C09127=1225.144,417.092,-82.048,-175.674,8.013,148.303
C09128=1225.147,416.687,-81.991,-175.674,8.010,148.302
C09129=1225.154,416.282,-81.934,-175.675,8.006,148.301
C09130=1225.160,415.877,-81.878,-175.676,8.003,148.301
C09131=1225.167,415.473,-81.820,-175.677,7.999,148.300
C09132=1225.171,415.226,-81.786,-175.678,7.997,148.300
C09133=1225.175,414.977,-81.752,-175.678,7.995,148.299
C09134=1225.180,414.730,-81.717,-175.679,7.993,148.299
C09135=1225.184,414.482,-81.682,-175.679,7.991,148.298
C09136=1225.188,414.235,-81.647,-175.679,7.988,148.298
C09137=1225.191,413.987,-81.613,-175.680,7.986,148.298
C09138=1225.196,413.740,-81.578,-175.681,7.985,148.297
C09139=1225.200,413.492,-81.544,-175.681,7.982,148.297
C09140=1225.204,413.244,-81.509,-175.682,7.979,148.296
C09141=1225.207,412.997,-81.474,-175.683,7.977,148.296
C09142=1225.212,412.750,-81.440,-175.683,7.975,148.295
C09143=1225.216,412.502,-81.405,-175.684,7.973,148.295
C09144=1225.220,412.254,-81.370,-175.684,7.971,148.295
C09145=1225.223,412.006,-81.336,-175.684,7.969,148.294
C09146=1225.228,411.759,-81.302,-175.685,7.967,148.294
C09147=1225.233,411.511,-81.267,-175.686,7.964,148.293
C09148=1225.236,411.264,-81.232,-175.686,7.962,148.293
C09149=1225.240,411.017,-81.198,-175.687,7.960,148.293
C09150=1225.244,410.769,-81.163,-175.688,7.958,148.292
C09151=1225.249,410.521,-81.129,-175.688,7.956,148.292
C09152=1225.252,410.274,-81.094,-175.688,7.954,148.291
C09153=1225.256,410.026,-81.060,-175.690,7.951,148.291
C09154=1225.260,409.778,-81.025,-175.690,7.949,148.290
C09155=1225.264,409.531,-80.991,-175.690,7.947,148.290
C09156=1225.269,409.283,-80.957,-175.691,7.945,148.290
C09157=1225.272,409.036,-80.921,-175.691,7.942,148.289
C09158=1225.277,408.789,-80.887,-175.692,7.940,148.289
C09159=1225.280,408.541,-80.852,-175.693,7.938,148.288
C09160=1225.285,408.293,-80.818,-175.693,7.935,148.288
C09161=1225.289,408.045,-80.783,-175.694,7.933,148.288
C09162=1225.293,407.798,-80.749,-175.695,7.931,148.287
C09163=1225.297,407.551,-80.715,-175.695,7.928,148.287
C09164=1225.301,407.303,-80.680,-175.696,7.926,148.286
C09165=1225.305,407.055,-80.646,-175.696,7.924,148.286
C09166=1225.309,406.807,-80.611,-175.697,7.922,148.285
C09167=1225.314,406.560,-80.577,-175.698,7.919,148.285
C09168=1225.317,406.313,-80.543,-175.698,7.917,148.284
C09169=1225.321,406.065,-80.508,-175.699,7.915,148.284
C09170=1225.325,405.818,-80.474,-175.699,7.913,148.284
C09171=1225.329,405.569,-80.439,-175.700,7.910,148.283
C09172=1225.334,405.322,-80.405,-175.701,7.908,148.283
C09173=1225.337,405.074,-80.371,-175.701,7.906,148.282
C09174=1225.342,404.827,-80.336,-175.702,7.904,148.282
C09175=1225.346,404.579,-80.302,-175.703,7.901,148.282
C09176=1225.349,404.332,-80.267,-175.703,7.899,148.281
C09177=1225.354,404.084,-80.233,-175.704,7.897,148.281
C09178=1225.358,403.837,-80.199,-175.705,7.894,148.280
C09179=1225.362,403.589,-80.164,-175.705,7.892,148.280
C09180=1225.366,403.341,-80.130,-175.706,7.889,148.279
C09181=1225.369,403.094,-80.096,-175.707,7.887,148.279
C09182=1225.374,402.846,-80.061,-175.707,7.885,148.279
C09183=1225.378,402.599,-80.027,-175.708,7.882,148.278
C09184=1225.382,402.350,-79.993,-175.709,7.880,148.278
C09185=1225.387,402.103,-79.959,-175.709,7.878,148.277
C09186=1225.391,401.856,-79.925,-175.710,7.875,148.277
C09187=1225.395,401.608,-79.890,-175.711,7.873,148.276
C09188=1225.398,401.361,-79.856,-175.711,7.871,148.276
C09189=1225.402,401.113,-79.821,-175.712,7.868,148.276
C09190=1225.406,400.865,-79.787,-175.713,7.865,148.275
C09191=1225.411,400.618,-79.753,-175.713,7.863,148.275
C09192=1225.415,400.370,-79.718,-175.714,7.861,148.274
C09193=1225.419,400.122,-79.685,-175.715,7.858,148.274
C09194=1225.423,399.875,-79.650,-175.715,7.856,148.273
C09195=1225.427,399.627,-79.616,-175.716,7.854,148.273
C09196=1225.431,399.379,-79.582,-175.717,7.851,148.273
C09197=1225.435,399.132,-79.548,-175.717,7.849,148.272
C09198=1225.439,398.884,-79.513,-175.719,7.846,148.272
C09199=1225.443,398.637,-79.480,-175.719,7.844,148.271
C09200=1225.448,398.389,-79.445,-175.719,7.842,148.271
C09201=1225.451,398.141,-79.411,-175.721,7.839,148.271
C09202=1225.456,397.894,-79.377,-175.721,7.837,148.270
C09203=1225.459,397.647,-79.343,-175.722,7.834,148.270
C09204=1225.464,397.398,-79.309,-175.723,7.832,148.269
C09205=1225.467,397.151,-79.275,-175.724,7.830,148.269
C09206=1225.472,396.904,-79.240,-175.724,7.827,148.268
C09207=1225.475,396.656,-79.206,-175.724,7.825,148.268
C09208=1225.480,396.408,-79.172,-175.726,7.822,148.268
C09209=1225.484,396.161,-79.139,-175.726,7.820,148.267
C09210=1225.489,395.913,-79.104,-175.727,7.817,148.267
C09211=1225.492,395.665,-79.070,-175.728,7.815,148.266
C09212=1225.497,395.417,-79.036,-175.729,7.813,148.266
C09213=1225.500,395.170,-79.002,-175.729,7.810,148.265
C09214=1225.504,394.922,-78.967,-175.730,7.807,148.265
C09215=1225.508,394.675,-78.934,-175.731,7.805,148.265
C09216=1225.513,394.427,-78.900,-175.732,7.803,148.264
C09217=1225.516,394.179,-78.866,-175.732,7.800,148.264
C09218=1225.521,393.932,-78.831,-175.733,7.798,148.263
C09219=1225.525,393.684,-78.798,-175.734,7.796,148.263
C09220=1225.529,393.403,-78.759,-175.735,7.792,148.262
C09221=1225.534,393.120,-78.720,-175.736,7.790,148.262
C09222=1225.539,392.840,-78.682,-175.737,7.787,148.261
C09223=1225.544,392.558,-78.644,-175.738,7.784,148.261
C09224=1225.548,392.310,-78.609,-175.738,7.782,148.261
C09225=1225.551,392.063,-78.575,-175.740,7.779,148.260
C09226=1225.556,391.815,-78.542,-175.740,7.777,148.260
C09227=1225.560,391.567,-78.507,-175.741,7.774,148.259
C09228=1225.563,391.320,-78.473,-175.742,7.772,148.259
C09229=1225.568,391.072,-78.439,-175.743,7.769,148.258
C09230=1225.572,390.824,-78.405,-175.744,7.766,148.258
C09231=1225.576,390.577,-78.372,-175.744,7.764,148.258
C09232=1225.580,390.329,-78.338,-175.745,7.761,148.257
C09233=1225.584,390.081,-78.304,-175.746,7.759,148.257
C09234=1225.589,389.833,-78.270,-175.747,7.756,148.256
C09235=1225.593,389.586,-78.236,-175.748,7.753,148.256
C09236=1225.596,389.338,-78.202,-175.749,7.752,148.256
C09237=1225.601,389.090,-78.168,-175.750,7.748,148.255
C09238=1225.605,388.843,-78.135,-175.750,7.746,148.255
C09239=1225.609,388.596,-78.101,-175.751,7.744,148.254
C09240=1225.613,388.347,-78.067,-175.753,7.741,148.254
C09241=1225.617,388.100,-78.033,-175.753,7.739,148.254
C09242=1225.621,387.852,-78.000,-175.754,7.736,148.253
C09243=1225.626,387.605,-77.965,-175.755,7.733,148.253
C09244=1225.630,387.357,-77.932,-175.756,7.731,148.252
C09245=1225.633,387.109,-77.898,-175.757,7.728,148.252
C09246=1225.638,386.861,-77.864,-175.758,7.725,148.251
C09247=1225.642,386.614,-77.830,-175.759,7.723,148.251
C09248=1225.646,386.366,-77.797,-175.760,7.720,148.251
C09249=1225.650,386.119,-77.763,-175.761,7.718,148.250
C09250=1225.654,385.870,-77.729,-175.762,7.716,148.250
C09251=1225.658,385.623,-77.695,-175.762,7.713,148.249
C09252=1225.662,385.376,-77.662,-175.764,7.710,148.249
C09253=1225.666,385.128,-77.628,-175.764,7.708,148.249
C09254=1225.671,384.880,-77.595,-175.765,7.705,148.248
C09255=1225.674,384.632,-77.561,-175.767,7.702,148.248
C09256=1225.678,384.385,-77.527,-175.767,7.700,148.247
C09257=1225.683,384.137,-77.493,-175.768,7.697,148.247
C09258=1225.687,383.890,-77.460,-175.770,7.694,148.247
C09259=1225.691,383.642,-77.426,-175.771,7.692,148.246
C09260=1225.695,383.394,-77.393,-175.771,7.690,148.246
C09261=1225.699,383.146,-77.358,-175.773,7.687,148.246
C09262=1225.703,382.898,-77.325,-175.774,7.684,148.245
C09263=1225.707,382.651,-77.292,-175.775,7.681,148.245
C09264=1225.711,382.404,-77.258,-175.775,7.679,148.244
C09265=1225.716,382.156,-77.224,-175.777,7.676,148.244
C09266=1225.720,381.908,-77.191,-175.778,7.674,148.244
C09267=1225.723,381.660,-77.157,-175.779,7.671,148.243
C09268=1225.727,381.412,-77.124,-175.780,7.669,148.243
C09269=1225.732,381.165,-77.091,-175.781,7.666,148.242
C09270=1225.736,380.917,-77.056,-175.782,7.663,148.242
C09271=1225.740,380.669,-77.023,-175.783,7.660,148.242
C09272=1225.744,380.422,-76.990,-175.784,7.657,148.241
C09273=1225.749,380.174,-76.957,-175.785,7.655,148.241
C09274=1225.752,379.926,-76.923,-175.786,7.653,148.241
C09275=1225.757,379.678,-76.889,-175.787,7.650,148.240
C09276=1225.761,379.430,-76.856,-175.788,7.647,148.240
C09277=1225.765,379.183,-76.823,-175.790,7.644,148.239
C09278=1225.769,378.936,-76.789,-175.791,7.641,148.239
C09279=1225.773,378.688,-76.756,-175.791,7.639,148.239
C09280=1225.777,378.440,-76.722,-175.793,7.637,148.238
C09281=1225.781,378.192,-76.689,-175.794,7.634,148.238
C09282=1225.786,377.944,-76.655,-175.795,7.631,148.237
C09283=1225.789,377.696,-76.621,-175.796,7.628,148.237
C09284=1225.793,377.449,-76.588,-175.797,7.625,148.237
C09285=1225.798,377.201,-76.555,-175.798,7.622,148.236
C09286=1225.802,376.953,-76.522,-175.800,7.621,148.236
C09287=1225.806,376.706,-76.489,-175.801,7.618,148.236
C09288=1225.810,376.458,-76.455,-175.802,7.615,148.235
C09289=1225.814,376.210,-76.422,-175.803,7.612,148.235
C09290=1225.818,375.963,-76.388,-175.804,7.609,148.234
C09291=1225.823,375.715,-76.355,-175.805,7.607,148.234
C09292=1225.827,375.467,-76.322,-175.807,7.604,148.234
C09293=1225.831,375.219,-76.288,-175.808,7.601,148.233
C09294=1225.835,374.972,-76.255,-175.809,7.598,148.233
C09295=1225.839,374.723,-76.222,-175.811,7.596,148.233
C09296=1225.843,374.476,-76.189,-175.811,7.594,148.232
C09297=1225.847,374.228,-76.155,-175.812,7.591,148.232
C09298=1225.851,373.980,-76.122,-175.814,7.588,148.232
C09299=1225.855,373.732,-76.089,-175.815,7.586,148.231
C09300=1225.859,373.485,-76.056,-175.816,7.583,148.231
C09301=1225.864,373.237,-76.023,-175.818,7.580,148.231
C09302=1225.868,372.989,-75.990,-175.819,7.577,148.230
C09303=1225.872,372.741,-75.956,-175.820,7.575,148.230
C09304=1225.876,372.494,-75.923,-175.821,7.572,148.230
C09305=1225.880,372.246,-75.890,-175.823,7.569,148.229
C09306=1225.884,371.998,-75.857,-175.824,7.566,148.229
C09307=1225.888,371.751,-75.824,-175.825,7.564,148.229
C09308=1225.893,371.503,-75.791,-175.827,7.561,148.228
C09309=1225.897,371.255,-75.757,-175.828,7.558,148.228
C09310=1225.901,371.007,-75.724,-175.829,7.555,148.228
C09311=1225.905,370.760,-75.691,-175.831,7.553,148.227
C09312=1225.909,370.512,-75.658,-175.832,7.550,148.227
C09313=1225.913,370.264,-75.625,-175.833,7.547,148.226
C09314=1225.917,370.016,-75.592,-175.835,7.544,148.226
C09315=1225.922,369.769,-75.559,-175.836,7.542,148.226
C09316=1225.926,369.521,-75.525,-175.837,7.539,148.226
C09317=1225.930,369.273,-75.492,-175.839,7.536,148.225
C09318=1225.934,369.025,-75.460,-175.840,7.533,148.225
C09319=1225.938,368.777,-75.427,-175.841,7.531,148.225
C09320=1225.942,368.530,-75.394,-175.843,7.528,148.224
C09321=1225.946,368.282,-75.361,-175.844,7.525,148.224
C09322=1225.950,368.034,-75.328,-175.845,7.523,148.224
C09323=1225.954,367.787,-75.295,-175.846,7.520,148.223
C09324=1225.959,367.506,-75.258,-175.849,7.516,148.223
C09325=1225.964,367.227,-75.220,-175.850,7.514,148.223
C09326=1225.968,366.947,-75.183,-175.852,7.510,148.222
C09327=1225.973,366.667,-75.146,-175.853,7.507,148.222
C09328=1225.977,366.420,-75.113,-175.854,7.505,148.222
C09329=1225.981,366.173,-75.081,-175.856,7.502,148.221
C09330=1225.985,365.925,-75.047,-175.857,7.499,148.221
C09331=1225.990,365.677,-75.015,-175.859,7.496,148.221
C09332=1225.994,365.429,-74.982,-175.860,7.493,148.220
C09333=1225.998,365.181,-74.949,-175.862,7.490,148.220
C09334=1226.002,364.934,-74.916,-175.863,7.488,148.220
C09335=1226.006,364.685,-74.884,-175.864,7.485,148.219
C09336=1226.010,364.438,-74.851,-175.866,7.482,148.219
C09337=1226.014,364.190,-74.817,-175.868,7.480,148.219
C09338=1226.019,363.941,-74.785,-175.869,7.477,148.219
C09339=1226.023,363.694,-74.752,-175.871,7.475,148.218
C09340=1226.026,363.446,-74.719,-175.872,7.471,148.218
C09341=1226.031,363.198,-74.687,-175.874,7.468,148.218
C09342=1226.035,362.950,-74.654,-175.875,7.465,148.217
C09343=1226.040,362.703,-74.621,-175.877,7.463,148.217
C09344=1226.043,362.455,-74.589,-175.878,7.460,148.217
C09345=1226.047,362.207,-74.556,-175.879,7.458,148.217
C09346=1226.052,361.960,-74.523,-175.881,7.455,148.216
C09347=1226.056,361.711,-74.490,-175.883,7.451,148.216
C09348=1226.059,361.464,-74.458,-175.884,7.449,148.216
C09349=1226.064,361.216,-74.425,-175.886,7.446,148.216
C09350=1226.068,360.968,-74.392,-175.887,7.444,148.215
C09351=1226.072,360.720,-74.360,-175.889,7.441,148.215
C09352=1226.076,360.473,-74.327,-175.890,7.438,148.215
C09353=1226.081,360.225,-74.294,-175.892,7.435,148.214
C09354=1226.085,359.977,-74.262,-175.894,7.432,148.214
C09355=1226.088,359.729,-74.229,-175.895,7.430,148.214
C09356=1226.093,359.481,-74.197,-175.897,7.427,148.214
C09357=1226.097,359.233,-74.164,-175.898,7.424,148.213
C09358=1226.101,358.985,-74.132,-175.900,7.422,148.213
C09359=1226.105,358.738,-74.099,-175.902,7.418,148.213
C09360=1226.110,358.490,-74.067,-175.903,7.416,148.213
C09361=1226.114,358.242,-74.035,-175.905,7.413,148.212
C09362=1226.118,357.994,-74.002,-175.906,7.411,148.212
C09363=1226.122,357.746,-73.969,-175.908,7.408,148.212
C09364=1226.126,357.498,-73.937,-175.910,7.404,148.212
C09365=1226.131,357.251,-73.905,-175.911,7.402,148.211
C09366=1226.135,357.003,-73.871,-175.913,7.399,148.211
C09367=1226.138,356.755,-73.840,-175.914,7.397,148.211
C09368=1226.143,356.506,-73.807,-175.916,7.394,148.211
C09369=1226.147,356.259,-73.774,-175.918,7.391,148.210
C09370=1226.151,356.011,-73.742,-175.920,7.388,148.210
C09371=1226.156,355.763,-73.710,-175.921,7.386,148.210
C09372=1226.159,355.516,-73.677,-175.922,7.383,148.210
C09373=1226.164,355.267,-73.645,-175.924,7.380,148.210
C09374=1226.168,355.020,-73.612,-175.926,7.377,148.209
C09375=1226.172,354.772,-73.580,-175.928,7.374,148.209
C09376=1226.177,354.524,-73.548,-175.930,7.372,148.209
C09377=1226.180,354.276,-73.516,-175.931,7.369,148.209
C09378=1226.184,354.028,-73.483,-175.933,7.366,148.208
C09379=1226.189,353.781,-73.451,-175.935,7.363,148.208
C09380=1226.193,353.532,-73.419,-175.936,7.361,148.208
C09381=1226.197,353.284,-73.387,-175.938,7.358,148.208
C09382=1226.201,353.037,-73.354,-175.939,7.356,148.208
C09383=1226.205,352.789,-73.323,-175.942,7.352,148.207
C09384=1226.210,352.541,-73.290,-175.943,7.350,148.207
C09385=1226.213,352.293,-73.258,-175.945,7.347,148.207
C09386=1226.218,352.045,-73.225,-175.947,7.345,148.207
C09387=1226.222,351.798,-73.194,-175.949,7.341,148.207
C09388=1226.226,351.550,-73.161,-175.950,7.338,148.206
C09389=1226.230,351.301,-73.129,-175.951,7.336,148.206
C09390=1226.234,351.053,-73.097,-175.953,7.333,148.206
C09391=1226.239,350.806,-73.065,-175.955,7.330,148.206
C09392=1226.243,350.558,-73.032,-175.957,7.327,148.205
C09393=1226.247,350.310,-73.000,-175.959,7.325,148.205
C09394=1226.252,350.062,-72.968,-175.960,7.322,148.205
C09395=1226.255,349.814,-72.936,-175.962,7.319,148.205
C09396=1226.260,349.566,-72.904,-175.964,7.317,148.205
C09397=1226.264,349.319,-72.873,-175.966,7.314,148.204
C09398=1226.269,349.070,-72.840,-175.967,7.311,148.204
C09399=1226.272,348.822,-72.808,-175.969,7.308,148.204
C09400=1226.276,348.574,-72.776,-175.971,7.306,148.204
C09401=1226.281,348.327,-72.744,-175.973,7.303,148.204
C09402=1226.285,348.079,-72.713,-175.974,7.301,148.203
C09403=1226.289,347.830,-72.680,-175.976,7.297,148.203
C09404=1226.294,347.583,-72.649,-175.979,7.295,148.203
C09405=1226.297,347.335,-72.617,-175.980,7.292,148.203
C09406=1226.302,347.087,-72.585,-175.982,7.289,148.203
C09407=1226.306,346.839,-72.553,-175.984,7.287,148.203
C09408=1226.310,346.591,-72.521,-175.986,7.284,148.202
C09409=1226.315,346.343,-72.489,-175.987,7.281,148.202
C09410=1226.318,346.095,-72.457,-175.989,7.278,148.202
C09411=1226.322,345.847,-72.425,-175.991,7.276,148.202
C09412=1226.327,345.600,-72.393,-175.993,7.273,148.202
C09413=1226.331,345.352,-72.361,-175.995,7.270,148.201
C09414=1226.335,345.104,-72.329,-175.997,7.267,148.202
C09415=1226.340,344.856,-72.297,-175.999,7.265,148.201
C09416=1226.343,344.608,-72.266,-176.000,7.262,148.201
C09417=1226.348,344.361,-72.234,-176.002,7.259,148.201
C09418=1226.352,344.112,-72.202,-176.004,7.256,148.201
C09419=1226.356,343.864,-72.170,-176.006,7.254,148.201
C09420=1226.360,343.616,-72.139,-176.008,7.251,148.200
C09421=1226.365,343.368,-72.107,-176.010,7.248,148.200
C09422=1226.369,343.121,-72.075,-176.012,7.246,148.200
C09423=1226.373,342.873,-72.043,-176.013,7.243,148.200
C09424=1226.377,342.625,-72.011,-176.015,7.240,148.200
C09425=1226.382,342.376,-71.980,-176.017,7.237,148.200
C09426=1226.386,342.128,-71.948,-176.019,7.235,148.200
C09427=1226.390,341.881,-71.917,-176.021,7.232,148.199
C09428=1226.394,341.603,-71.881,-176.023,7.229,148.199
C09429=1226.400,341.325,-71.846,-176.025,7.226,148.199
C09430=1226.404,341.047,-71.810,-176.028,7.223,148.199
C09431=1226.409,340.770,-71.775,-176.029,7.220,148.199
C09432=1226.413,340.522,-71.744,-176.032,7.217,148.199
C09433=1226.417,340.274,-71.712,-176.033,7.214,148.198
C09434=1226.422,340.026,-71.680,-176.035,7.212,148.198
C09435=1226.426,339.778,-71.649,-176.037,7.209,148.198
C09436=1226.430,339.530,-71.617,-176.039,7.206,148.198
C09437=1226.434,339.282,-71.585,-176.041,7.204,148.198
C09438=1226.438,339.034,-71.555,-176.043,7.201,148.198
C09439=1226.442,338.786,-71.523,-176.045,7.198,148.198
C09440=1226.447,338.538,-71.492,-176.047,7.196,148.197
C09441=1226.451,338.290,-71.459,-176.049,7.193,148.197
C09442=1226.455,338.043,-71.428,-176.051,7.190,148.197
C09443=1226.459,337.794,-71.397,-176.053,7.188,148.197
C09444=1226.464,337.547,-71.365,-176.055,7.185,148.197
C09445=1226.468,337.298,-71.334,-176.057,7.182,148.197
C09446=1226.472,337.051,-71.303,-176.059,7.180,148.197
C09447=1226.476,336.802,-71.271,-176.061,7.177,148.197
C09448=1226.480,336.555,-71.240,-176.063,7.174,148.197
C09449=1226.484,336.306,-71.208,-176.065,7.172,148.197
C09450=1226.489,336.059,-71.178,-176.066,7.169,148.196
C09451=1226.492,335.810,-71.146,-176.069,7.166,148.196
C09452=1226.497,335.563,-71.115,-176.071,7.164,148.196
C09453=1226.501,335.314,-71.083,-176.072,7.161,148.196
C09454=1226.506,335.066,-71.052,-176.075,7.158,148.196
C09455=1226.510,334.818,-71.020,-176.077,7.155,148.196
C09456=1226.514,334.570,-70.989,-176.078,7.153,148.196
C09457=1226.518,334.322,-70.958,-176.081,7.150,148.196
C09458=1226.523,334.074,-70.927,-176.083,7.147,148.195
C09459=1226.527,333.826,-70.896,-176.085,7.145,148.195
C09460=1226.531,333.578,-70.864,-176.087,7.142,148.195
C09461=1226.536,333.330,-70.833,-176.089,7.139,148.195
C09462=1226.540,333.082,-70.802,-176.091,7.137,148.195
C09463=1226.544,332.834,-70.771,-176.093,7.134,148.195
C09464=1226.547,332.586,-70.740,-176.095,7.131,148.195
C09465=1226.551,332.339,-70.709,-176.096,7.129,148.195
C09466=1226.556,332.091,-70.678,-176.099,7.126,148.195
C09467=1226.560,331.842,-70.647,-176.101,7.123,148.195
C09468=1226.564,331.595,-70.615,-176.103,7.121,148.195
C09469=1226.568,331.346,-70.584,-176.105,7.118,148.194
C09470=1226.573,331.098,-70.553,-176.107,7.115,148.194
C09471=1226.578,330.850,-70.522,-176.109,7.113,148.194
C09472=1226.581,330.602,-70.491,-176.111,7.110,148.194
C09473=1226.586,330.354,-70.460,-176.113,7.107,148.194
C09474=1226.590,330.105,-70.429,-176.115,7.105,148.194
C09475=1226.595,329.857,-70.398,-176.117,7.102,148.194
C09476=1226.599,329.610,-70.366,-176.119,7.099,148.194
C09477=1226.602,329.362,-70.336,-176.121,7.097,148.194
C09478=1226.607,329.114,-70.305,-176.124,7.094,148.194
C09479=1226.611,328.866,-70.274,-176.126,7.092,148.194
C09480=1226.615,328.618,-70.243,-176.127,7.089,148.194
C09481=1226.620,328.370,-70.212,-176.130,7.086,148.194
C09482=1226.624,328.122,-70.181,-176.132,7.084,148.193
C09483=1226.628,327.873,-70.150,-176.134,7.081,148.193
C09484=1226.632,327.626,-70.120,-176.136,7.078,148.193
C09485=1226.637,327.378,-70.089,-176.138,7.076,148.193
C09486=1226.641,327.129,-70.058,-176.140,7.074,148.193
C09487=1226.645,326.882,-70.026,-176.142,7.070,148.193
C09488=1226.650,326.634,-69.996,-176.144,7.068,148.193
C09489=1226.653,326.385,-69.965,-176.147,7.066,148.193
C09490=1226.658,326.137,-69.934,-176.149,7.062,148.193
C09491=1226.662,325.889,-69.904,-176.151,7.060,148.193
C09492=1226.666,325.641,-69.872,-176.152,7.058,148.193
C09493=1226.670,325.393,-69.842,-176.155,7.055,148.193
C09494=1226.675,325.145,-69.811,-176.157,7.052,148.193
C09495=1226.679,324.896,-69.780,-176.159,7.050,148.193
C09496=1226.683,324.649,-69.750,-176.161,7.047,148.193
C09497=1226.687,324.401,-69.719,-176.164,7.044,148.193
C09498=1226.692,324.153,-69.689,-176.165,7.042,148.193
C09499=1226.696,323.904,-69.658,-176.168,7.039,148.193
C09500=1226.700,323.657,-69.627,-176.170,7.037,148.193
C09501=1226.704,323.409,-69.597,-176.172,7.034,148.192
C09502=1226.709,323.161,-69.566,-176.174,7.031,148.192
C09503=1226.713,322.912,-69.535,-176.176,7.029,148.192
C09504=1226.717,322.664,-69.505,-176.178,7.027,148.193
C09505=1226.721,322.416,-69.474,-176.181,7.023,148.192
C09506=1226.726,322.168,-69.443,-176.183,7.021,148.192
C09507=1226.730,321.919,-69.413,-176.185,7.019,148.192
C09508=1226.734,321.672,-69.382,-176.187,7.015,148.192
C09509=1226.738,321.424,-69.352,-176.189,7.013,148.192
C09510=1226.743,321.176,-69.322,-176.191,7.011,148.192
C09511=1226.747,320.927,-69.290,-176.194,7.008,148.192
C09512=1226.751,320.680,-69.260,-176.196,7.005,148.192
C09513=1226.756,320.431,-69.230,-176.198,7.003,148.192
C09514=1226.760,320.183,-69.199,-176.200,7.000,148.192
C09515=1226.763,319.935,-69.169,-176.202,6.998,148.192
C09516=1226.768,319.687,-69.138,-176.204,6.995,148.192
C09517=1226.772,319.439,-69.108,-176.207,6.992,148.192
C09518=1226.777,319.191,-69.078,-176.209,6.990,148.192
C09519=1226.781,318.943,-69.048,-176.211,6.988,148.192
C09520=1226.785,318.695,-69.017,-176.214,6.985,148.192
C09521=1226.789,318.446,-68.986,-176.215,6.982,148.192
C09522=1226.794,318.198,-68.956,-176.217,6.980,148.192
C09523=1226.798,317.950,-68.926,-176.220,6.977,148.192
C09524=1226.802,317.702,-68.895,-176.222,6.975,148.192
C09525=1226.807,317.454,-68.865,-176.224,6.973,148.192
C09526=1226.811,317.206,-68.835,-176.226,6.969,148.192
C09527=1226.815,316.958,-68.804,-176.228,6.967,148.192
C09528=1226.819,316.709,-68.775,-176.230,6.965,148.192
C09529=1226.824,316.461,-68.744,-176.233,6.962,148.192
C09530=1226.828,316.214,-68.714,-176.235,6.960,148.192
C09531=1226.832,315.965,-68.684,-176.237,6.957,148.192
C09532=1226.836,315.690,-68.650,-176.240,6.954,148.192
C09533=1226.842,315.413,-68.616,-176.242,6.951,148.192
C09534=1226.846,315.138,-68.583,-176.245,6.948,148.192
C09535=1226.851,314.862,-68.550,-176.247,6.946,148.192
C09536=1226.855,314.614,-68.519,-176.250,6.943,148.192
C09537=1226.860,314.366,-68.489,-176.252,6.940,148.192
C09538=1226.864,314.118,-68.459,-176.254,6.938,148.192
C09539=1226.868,313.869,-68.429,-176.256,6.935,148.192
C09540=1226.872,313.621,-68.399,-176.259,6.933,148.192
C09541=1226.876,313.373,-68.369,-176.261,6.931,148.192
C09542=1226.881,313.125,-68.338,-176.263,6.928,148.192
C09543=1226.885,312.877,-68.309,-176.265,6.925,148.192
C09544=1226.890,312.629,-68.278,-176.267,6.923,148.192
C09545=1226.894,312.381,-68.249,-176.270,6.920,148.192
C09546=1226.898,312.133,-68.218,-176.272,6.917,148.192
C09547=1226.903,311.884,-68.188,-176.274,6.915,148.192
C09548=1226.907,311.637,-68.158,-176.277,6.912,148.192
C09549=1226.911,311.388,-68.129,-176.279,6.910,148.192
C09550=1226.916,311.140,-68.099,-176.281,6.908,148.192
C09551=1226.920,310.892,-68.069,-176.283,6.906,148.192
C09552=1226.924,310.644,-68.039,-176.286,6.902,148.192
C09553=1226.929,310.395,-68.009,-176.288,6.900,148.192
C09554=1226.933,310.148,-67.979,-176.290,6.898,148.192
C09555=1226.936,309.899,-67.949,-176.292,6.895,148.192
C09556=1226.941,309.650,-67.919,-176.295,6.893,148.192
C09557=1226.945,309.402,-67.889,-176.297,6.891,148.192
C09558=1226.949,309.154,-67.859,-176.299,6.887,148.192
C09559=1226.954,308.906,-67.829,-176.301,6.885,148.192
C09560=1226.958,308.658,-67.799,-176.303,6.883,148.192
C09561=1226.962,308.410,-67.770,-176.306,6.880,148.192
C09562=1226.966,308.161,-67.740,-176.308,6.878,148.193
C09563=1226.971,307.913,-67.710,-176.310,6.876,148.193
C09564=1226.975,307.665,-67.680,-176.313,6.873,148.193
C09565=1226.979,307.417,-67.651,-176.315,6.870,148.193
C09566=1226.984,307.169,-67.622,-176.317,6.868,148.193
C09567=1226.989,306.921,-67.592,-176.320,6.865,148.193
C09568=1226.993,306.673,-67.562,-176.322,6.863,148.193
C09569=1226.997,306.425,-67.532,-176.324,6.861,148.193
C09570=1227.001,306.177,-67.502,-176.327,6.858,148.193
C09571=1227.005,305.928,-67.473,-176.329,6.855,148.193
C09572=1227.010,305.680,-67.443,-176.331,6.853,148.193
C09573=1227.014,305.431,-67.413,-176.333,6.851,148.193
C09574=1227.019,305.183,-67.384,-176.336,6.848,148.193
C09575=1227.023,304.935,-67.355,-176.338,6.846,148.193
C09576=1227.027,304.687,-67.324,-176.340,6.843,148.193
C09577=1227.031,304.439,-67.295,-176.343,6.840,148.193
C09578=1227.035,304.191,-67.266,-176.345,6.838,148.193
C09579=1227.040,303.942,-67.235,-176.347,6.836,148.193
C09580=1227.044,303.694,-67.206,-176.350,6.833,148.193
C09581=1227.048,303.446,-67.177,-176.352,6.831,148.193
C09582=1227.053,303.198,-67.147,-176.354,6.829,148.194
C09583=1227.057,302.950,-67.118,-176.356,6.826,148.194
C09584=1227.062,302.702,-67.089,-176.359,6.823,148.194
C09585=1227.066,302.453,-67.059,-176.361,6.821,148.194
C09586=1227.070,302.205,-67.030,-176.363,6.819,148.194
C09587=1227.074,301.957,-67.000,-176.366,6.816,148.194
C09588=1227.078,301.708,-66.971,-176.368,6.814,148.194
C09589=1227.082,301.460,-66.941,-176.370,6.812,148.194
C09590=1227.087,301.212,-66.911,-176.373,6.809,148.194
C09591=1227.092,300.964,-66.882,-176.375,6.807,148.194
C09592=1227.096,300.716,-66.853,-176.377,6.804,148.194
C09593=1227.101,300.467,-66.824,-176.379,6.802,148.194
C09594=1227.105,300.219,-66.795,-176.382,6.799,148.194
C09595=1227.109,299.970,-66.765,-176.384,6.797,148.194
C09596=1227.113,299.722,-66.736,-176.386,6.795,148.194
C09597=1227.118,299.474,-66.706,-176.389,6.792,148.195
C09598=1227.122,299.226,-66.677,-176.392,6.790,148.195
C09599=1227.126,298.978,-66.648,-176.394,6.787,148.195
C09600=1227.131,298.729,-66.619,-176.396,6.785,148.195
C09601=1227.135,298.481,-66.589,-176.398,6.782,148.195
C09602=1227.139,298.233,-66.560,-176.401,6.780,148.195
C09603=1227.143,297.985,-66.531,-176.403,6.778,148.195
C09604=1227.148,297.737,-66.502,-176.406,6.775,148.195
C09605=1227.152,297.488,-66.473,-176.408,6.773,148.195
C09606=1227.156,297.240,-66.444,-176.410,6.771,148.195
C09607=1227.160,296.992,-66.414,-176.412,6.768,148.195
C09608=1227.165,296.743,-66.385,-176.415,6.766,148.196
C09609=1227.170,296.495,-66.357,-176.417,6.763,148.196
C09610=1227.174,296.247,-66.327,-176.419,6.761,148.196
C09611=1227.178,295.999,-66.298,-176.422,6.758,148.196
C09612=1227.183,295.750,-66.269,-176.424,6.756,148.196
C09613=1227.187,295.503,-66.240,-176.427,6.754,148.196
C09614=1227.191,295.254,-66.211,-176.429,6.752,148.196
C09615=1227.195,295.005,-66.182,-176.432,6.749,148.196
C09616=1227.199,294.757,-66.153,-176.434,6.746,148.196
C09617=1227.204,294.510,-66.124,-176.436,6.745,148.196
C09618=1227.209,294.261,-66.095,-176.438,6.742,148.196
C09619=1227.213,294.012,-66.065,-176.441,6.739,148.196
C09620=1227.216,293.764,-66.037,-176.443,6.737,148.197
C09621=1227.221,293.516,-66.008,-176.446,6.735,148.197
C09622=1227.226,293.268,-65.979,-176.448,6.733,148.197
C09623=1227.230,293.019,-65.950,-176.451,6.730,148.197
C09624=1227.234,292.771,-65.921,-176.453,6.728,148.197
C09625=1227.239,292.523,-65.893,-176.455,6.726,148.197
C09626=1227.243,292.275,-65.863,-176.458,6.723,148.197
C09627=1227.247,292.026,-65.835,-176.460,6.721,148.197
C09628=1227.252,291.778,-65.806,-176.462,6.718,148.197
C09629=1227.256,291.530,-65.777,-176.465,6.716,148.198
C09630=1227.260,291.281,-65.748,-176.467,6.713,148.198
C09631=1227.264,291.032,-65.719,-176.470,6.711,148.198
C09632=1227.269,290.785,-65.690,-176.472,6.709,148.198
C09633=1227.273,290.536,-65.662,-176.474,6.707,148.198
C09634=1227.277,290.288,-65.633,-176.477,6.704,148.198
C09635=1227.282,290.040,-65.604,-176.479,6.702,148.198
C09636=1227.287,289.766,-65.573,-176.482,6.700,148.198
C09637=1227.292,289.492,-65.540,-176.484,6.697,148.198
C09638=1227.296,289.217,-65.509,-176.487,6.694,148.199
C09639=1227.301,288.943,-65.477,-176.489,6.692,148.199
C09640=1227.306,288.695,-65.449,-176.492,6.690,148.199
C09641=1227.310,288.447,-65.420,-176.495,6.687,148.199
C09642=1227.315,288.199,-65.391,-176.497,6.685,148.199
C09643=1227.319,287.950,-65.363,-176.499,6.683,148.199
C09644=1227.323,287.702,-65.334,-176.502,6.681,148.199
C09645=1227.327,287.454,-65.306,-176.504,6.678,148.199
C09646=1227.332,287.205,-65.277,-176.507,6.676,148.200
C09647=1227.336,286.957,-65.248,-176.509,6.673,148.200
C09648=1227.340,286.709,-65.220,-176.511,6.671,148.200
C09649=1227.345,286.460,-65.191,-176.514,6.669,148.200
C09650=1227.350,286.212,-65.163,-176.516,6.666,148.200
C09651=1227.353,285.964,-65.134,-176.518,6.664,148.200
C09652=1227.358,285.715,-65.105,-176.521,6.662,148.201
C09653=1227.362,285.467,-65.077,-176.523,6.660,148.201
C09654=1227.366,285.218,-65.049,-176.526,6.657,148.201
C09655=1227.371,284.970,-65.021,-176.528,6.655,148.201
C09656=1227.375,284.722,-64.991,-176.530,6.653,148.201
C09657=1227.379,284.473,-64.963,-176.533,6.651,148.201
C09658=1227.384,284.225,-64.935,-176.535,6.649,148.201
C09659=1227.388,283.977,-64.906,-176.538,6.646,148.201
C09660=1227.393,283.729,-64.878,-176.540,6.644,148.202
C09661=1227.397,283.480,-64.850,-176.543,6.641,148.202
C09662=1227.401,283.232,-64.822,-176.545,6.640,148.202
C09663=1227.406,282.983,-64.793,-176.548,6.637,148.202
C09664=1227.410,282.736,-64.765,-176.550,6.634,148.202
C09665=1227.415,282.487,-64.736,-176.553,6.632,148.202
C09666=1227.419,282.239,-64.708,-176.555,6.630,148.202
C09667=1227.423,281.990,-64.679,-176.557,6.628,148.203
C09668=1227.428,281.742,-64.652,-176.560,6.625,148.203
C09669=1227.432,281.493,-64.623,-176.562,6.623,148.203
C09670=1227.436,281.245,-64.595,-176.565,6.621,148.203
C09671=1227.440,280.997,-64.567,-176.567,6.619,148.203
C09672=1227.445,280.748,-64.538,-176.569,6.617,148.203
C09673=1227.449,280.500,-64.511,-176.572,6.614,148.203
C09674=1227.454,280.251,-64.482,-176.575,6.612,148.204
C09675=1227.458,280.003,-64.454,-176.577,6.610,148.204
C09676=1227.462,279.755,-64.426,-176.579,6.608,148.204
C09677=1227.467,279.507,-64.397,-176.581,6.606,148.204
C09678=1227.471,279.259,-64.370,-176.584,6.603,148.204
C09679=1227.476,279.010,-64.341,-176.587,6.601,148.204
C09680=1227.480,278.761,-64.314,-176.589,6.599,148.205
C09681=1227.484,278.513,-64.286,-176.591,6.597,148.205
C09682=1227.489,278.265,-64.257,-176.593,6.594,148.205
C09683=1227.493,278.016,-64.229,-176.596,6.593,148.205
C09684=1227.497,277.768,-64.201,-176.599,6.590,148.205
C09685=1227.502,277.519,-64.173,-176.601,6.588,148.206
C09686=1227.506,277.271,-64.145,-176.603,6.585,148.206
C09687=1227.510,277.022,-64.118,-176.606,6.584,148.206
C09688=1227.515,276.774,-64.089,-176.608,6.581,148.206
C09689=1227.520,276.526,-64.061,-176.611,6.579,148.206
C09690=1227.523,276.278,-64.033,-176.613,6.576,148.206
C09691=1227.528,276.029,-64.005,-176.616,6.574,148.207
C09692=1227.532,275.780,-63.977,-176.618,6.572,148.207
C09693=1227.537,275.532,-63.950,-176.621,6.570,148.207
C09694=1227.541,275.284,-63.922,-176.623,6.568,148.207
C09695=1227.546,275.036,-63.893,-176.626,6.565,148.207
C09696=1227.550,274.787,-63.866,-176.628,6.563,148.207
C09697=1227.554,274.538,-63.838,-176.631,6.561,148.208
C09698=1227.558,274.291,-63.810,-176.633,6.559,148.208
C09699=1227.563,274.042,-63.781,-176.635,6.557,148.208
C09700=1227.568,273.793,-63.754,-176.638,6.555,148.208
C09701=1227.572,273.545,-63.727,-176.641,6.552,148.208
C09702=1227.576,273.297,-63.698,-176.643,6.550,148.208
C09703=1227.581,273.048,-63.671,-176.645,6.548,148.209
C09704=1227.585,272.800,-63.643,-176.648,6.546,148.209
C09705=1227.589,272.551,-63.616,-176.650,6.544,148.209
C09706=1227.594,272.303,-63.588,-176.652,6.542,148.209
C09707=1227.598,272.055,-63.560,-176.655,6.540,148.209
C09708=1227.602,271.806,-63.533,-176.658,6.537,148.209
C09709=1227.607,271.558,-63.504,-176.660,6.535,148.210
C09710=1227.612,271.309,-63.477,-176.662,6.533,148.210
C09711=1227.616,271.061,-63.449,-176.665,6.531,148.210
C09712=1227.620,270.813,-63.421,-176.667,6.529,148.210
C09713=1227.625,270.564,-63.394,-176.670,6.527,148.210
C09714=1227.628,270.316,-63.366,-176.672,6.525,148.211
C09715=1227.633,270.067,-63.339,-176.675,6.522,148.211
C09716=1227.638,269.819,-63.311,-176.677,6.520,148.211
C09717=1227.642,269.570,-63.283,-176.680,6.518,148.211
C09718=1227.647,269.322,-63.255,-176.682,6.516,148.211
C09719=1227.651,269.073,-63.228,-176.684,6.514,148.212
C09720=1227.655,268.824,-63.201,-176.687,6.512,148.212
C09721=1227.660,268.576,-63.173,-176.689,6.510,148.212
C09722=1227.664,268.328,-63.146,-176.692,6.507,148.212
C09723=1227.669,268.080,-63.118,-176.695,6.505,148.212
C09724=1227.673,267.831,-63.091,-176.697,6.503,148.213
C09725=1227.677,267.583,-63.063,-176.699,6.501,148.213
C09726=1227.682,267.334,-63.036,-176.702,6.499,148.213
C09727=1227.686,267.086,-63.009,-176.704,6.497,148.213
C09728=1227.690,266.837,-62.981,-176.707,6.495,148.213
C09729=1227.695,266.589,-62.954,-176.709,6.493,148.214
C09730=1227.699,266.340,-62.927,-176.712,6.490,148.214
C09731=1227.704,266.092,-62.899,-176.714,6.488,148.214
C09732=1227.708,265.843,-62.872,-176.717,6.486,148.214
C09733=1227.713,265.595,-62.844,-176.719,6.484,148.214
C09734=1227.717,265.347,-62.817,-176.722,6.482,148.215
C09735=1227.722,265.098,-62.790,-176.724,6.480,148.215
C09736=1227.726,264.849,-62.762,-176.726,6.478,148.215
C09737=1227.730,264.601,-62.735,-176.729,6.476,148.215
C09738=1227.735,264.353,-62.707,-176.731,6.474,148.216
C09739=1227.739,264.104,-62.680,-176.734,6.472,148.216
C09740=1227.745,263.832,-62.650,-176.737,6.469,148.216
C09741=1227.749,263.559,-62.620,-176.739,6.467,148.216
C09742=1227.754,263.287,-62.591,-176.742,6.464,148.216
C09743=1227.759,263.013,-62.561,-176.745,6.462,148.216
C09744=1227.763,262.765,-62.534,-176.747,6.460,148.217
C09745=1227.768,262.517,-62.506,-176.750,6.458,148.217
C09746=1227.771,262.269,-62.479,-176.752,6.456,148.217
C09747=1227.776,262.020,-62.452,-176.755,6.454,148.217
C09748=1227.781,261.772,-62.425,-176.758,6.452,148.218
C09749=1227.785,261.522,-62.398,-176.760,6.449,148.218
C09750=1227.790,261.274,-62.371,-176.762,6.447,148.218
C09751=1227.794,261.025,-62.344,-176.765,6.446,148.218
C09752=1227.799,260.778,-62.316,-176.767,6.443,148.218
C09753=1227.802,260.529,-62.289,-176.770,6.441,148.219
C09754=1227.807,260.281,-62.262,-176.772,6.440,148.219
C09755=1227.812,260.032,-62.235,-176.774,6.437,148.219
C09756=1227.816,259.783,-62.208,-176.777,6.435,148.219
C09757=1227.820,259.535,-62.181,-176.780,6.434,148.220
C09758=1227.824,259.287,-62.154,-176.782,6.431,148.220
C09759=1227.829,259.038,-62.127,-176.784,6.429,148.220
C09760=1227.834,258.790,-62.100,-176.787,6.428,148.220
C09761=1227.838,258.541,-62.073,-176.790,6.425,148.221
C09762=1227.843,258.293,-62.046,-176.792,6.423,148.221
C09763=1227.847,258.044,-62.020,-176.795,6.421,148.221
C09764=1227.852,257.796,-61.993,-176.797,6.419,148.221
C09765=1227.856,257.547,-61.965,-176.800,6.417,148.221
C09766=1227.860,257.298,-61.938,-176.802,6.415,148.222
C09767=1227.864,257.050,-61.912,-176.804,6.413,148.222
C09768=1227.869,256.801,-61.885,-176.807,6.411,148.222
C09769=1227.874,256.552,-61.858,-176.810,6.409,148.222
C09770=1227.878,256.304,-61.832,-176.812,6.407,148.223
C09771=1227.882,256.056,-61.805,-176.814,6.405,148.223
C09772=1227.887,255.807,-61.778,-176.817,6.403,148.223
C09773=1227.892,255.559,-61.750,-176.820,6.401,148.223
C09774=1227.896,255.311,-61.724,-176.822,6.399,148.224
C09775=1227.900,255.062,-61.697,-176.824,6.397,148.224
C09776=1227.905,254.813,-61.671,-176.827,6.395,148.224
C09777=1227.909,254.565,-61.644,-176.829,6.393,148.224
C09778=1227.914,254.316,-61.617,-176.832,6.390,148.225
C09779=1227.918,254.068,-61.590,-176.835,6.388,148.225
C09780=1227.922,253.820,-61.564,-176.837,6.386,148.225
C09781=1227.927,253.570,-61.537,-176.840,6.384,148.225
C09782=1227.931,253.322,-61.511,-176.842,6.382,148.226
C09783=1227.936,253.074,-61.484,-176.845,6.380,148.226
C09784=1227.941,252.825,-61.457,-176.847,6.378,148.226
C09785=1227.945,252.576,-61.431,-176.849,6.376,148.226
C09786=1227.949,252.328,-61.404,-176.852,6.374,148.227
C09787=1227.953,252.080,-61.377,-176.855,6.372,148.227
C09788=1227.958,251.831,-61.351,-176.857,6.370,148.227
C09789=1227.963,251.582,-61.324,-176.859,6.368,148.227
C09790=1227.967,251.334,-61.297,-176.862,6.367,148.228
C09791=1227.972,251.085,-61.270,-176.865,6.365,148.228
C09792=1227.976,250.837,-61.245,-176.867,6.362,148.228
C09793=1227.980,250.588,-61.218,-176.869,6.361,148.228
C09794=1227.985,250.339,-61.192,-176.872,6.359,148.229
C09795=1227.989,250.091,-61.165,-176.875,6.357,148.229
C09796=1227.993,249.843,-61.138,-176.877,6.355,148.229
C09797=1227.998,249.594,-61.112,-176.879,6.353,148.229
C09798=1228.002,249.345,-61.086,-176.882,6.351,148.230
C09799=1228.007,249.096,-61.059,-176.885,6.349,148.230
C09800=1228.011,248.848,-61.033,-176.887,6.347,148.230
C09801=1228.016,248.600,-61.006,-176.889,6.345,148.230
C09802=1228.020,248.351,-60.980,-176.892,6.343,148.231
C09803=1228.025,248.102,-60.953,-176.895,6.341,148.231
C09804=1228.029,247.854,-60.927,-176.897,6.339,148.231
C09805=1228.034,247.606,-60.900,-176.899,6.337,148.231
C09806=1228.038,247.357,-60.875,-176.902,6.335,148.232
C09807=1228.043,247.108,-60.848,-176.904,6.333,148.232
C09808=1228.047,246.860,-60.822,-176.907,6.331,148.232
C09809=1228.051,246.611,-60.795,-176.909,6.329,148.232
C09810=1228.056,246.362,-60.769,-176.912,6.327,148.233
C09811=1228.060,246.113,-60.743,-176.914,6.325,148.233
C09812=1228.065,245.865,-60.716,-176.917,6.324,148.233
C09813=1228.069,245.616,-60.690,-176.920,6.322,148.234
C09814=1228.074,245.369,-60.664,-176.922,6.319,148.234
C09815=1228.079,245.120,-60.638,-176.924,6.318,148.234
C09816=1228.083,244.871,-60.612,-176.927,6.316,148.234
C09817=1228.088,244.622,-60.585,-176.930,6.314,148.235
C09818=1228.092,244.373,-60.559,-176.932,6.312,148.235
C09819=1228.096,244.125,-60.533,-176.934,6.310,148.235
C09820=1228.101,243.876,-60.507,-176.937,6.308,148.235
C09821=1228.105,243.628,-60.481,-176.940,6.306,148.236
C09822=1228.109,243.380,-60.455,-176.942,6.304,148.236
C09823=1228.114,243.131,-60.428,-176.945,6.302,148.236
C09824=1228.119,242.882,-60.403,-176.947,6.300,148.236
C09825=1228.123,242.633,-60.377,-176.950,6.298,148.237
C09826=1228.128,242.385,-60.350,-176.952,6.296,148.237
C09827=1228.132,242.137,-60.324,-176.955,6.294,148.237
C09828=1228.136,241.888,-60.299,-176.957,6.292,148.238
C09829=1228.141,241.639,-60.273,-176.960,6.290,148.238
C09830=1228.145,241.390,-60.246,-176.962,6.288,148.238
C09831=1228.150,241.142,-60.220,-176.965,6.287,148.238
C09832=1228.154,240.894,-60.195,-176.967,6.285,148.239
C09833=1228.159,240.645,-60.169,-176.970,6.283,148.239
C09834=1228.163,240.396,-60.142,-176.973,6.281,148.239
C09835=1228.168,240.147,-60.116,-176.975,6.279,148.239
C09836=1228.172,239.899,-60.091,-176.977,6.277,148.240
C09837=1228.177,239.651,-60.065,-176.979,6.276,148.240
C09838=1228.182,239.401,-60.039,-176.982,6.274,148.240
C09839=1228.186,239.153,-60.013,-176.985,6.272,148.241
C09840=1228.191,238.905,-59.988,-176.987,6.270,148.241
C09841=1228.195,238.656,-59.961,-176.990,6.268,148.241
C09842=1228.199,238.408,-59.935,-176.992,6.266,148.241
C09843=1228.204,238.158,-59.909,-176.995,6.264,148.242
C09844=1228.209,237.887,-59.881,-176.997,6.262,148.242
C09845=1228.214,237.615,-59.853,-177.000,6.260,148.242
C09846=1228.219,237.345,-59.825,-177.003,6.258,148.243
C09847=1228.223,237.073,-59.797,-177.006,6.256,148.243
C09848=1228.228,236.824,-59.771,-177.008,6.254,148.243
C09849=1228.232,236.576,-59.746,-177.011,6.252,148.244
C09850=1228.237,236.327,-59.720,-177.014,6.250,148.244
C09851=1228.241,236.078,-59.694,-177.016,6.248,148.244
C09852=1228.245,235.830,-59.669,-177.019,6.246,148.244
C09853=1228.251,235.581,-59.643,-177.021,6.245,148.245
C09854=1228.255,235.332,-59.617,-177.024,6.242,148.245
C09855=1228.259,235.083,-59.591,-177.026,6.241,148.245
C09856=1228.264,234.835,-59.566,-177.029,6.239,148.246
C09857=1228.268,234.587,-59.540,-177.031,6.238,148.246
C09858=1228.272,234.338,-59.514,-177.033,6.236,148.246
C09859=1228.277,234.090,-59.489,-177.036,6.234,148.246
C09860=1228.281,233.841,-59.463,-177.039,6.232,148.247
C09861=1228.286,233.592,-59.437,-177.041,6.230,148.247
C09862=1228.291,233.343,-59.413,-177.044,6.228,148.247
C09863=1228.295,233.095,-59.387,-177.046,6.226,148.248
C09864=1228.299,232.846,-59.361,-177.049,6.224,148.248
C09865=1228.304,232.598,-59.336,-177.051,6.222,148.248
C09866=1228.308,232.349,-59.310,-177.054,6.220,148.249
C09867=1228.313,232.100,-59.284,-177.057,6.219,148.249
C09868=1228.317,231.852,-59.259,-177.059,6.217,148.249
C09869=1228.322,231.602,-59.234,-177.062,6.215,148.249
C09870=1228.327,231.354,-59.208,-177.064,6.214,148.250
C09871=1228.331,231.106,-59.183,-177.066,6.212,148.250
C09872=1228.335,230.857,-59.157,-177.069,6.210,148.250
C09873=1228.340,230.608,-59.132,-177.071,6.208,148.251
C09874=1228.344,230.359,-59.106,-177.074,6.206,148.251
C09875=1228.349,230.111,-59.081,-177.076,6.204,148.251
C09876=1228.354,229.862,-59.055,-177.079,6.202,148.252
C09877=1228.358,229.613,-59.030,-177.082,6.200,148.252
C09878=1228.363,229.365,-59.005,-177.084,6.198,148.252
C09879=1228.367,229.116,-58.979,-177.087,6.197,148.252
C09880=1228.372,228.868,-58.954,-177.090,6.195,148.253
C09881=1228.376,228.618,-58.929,-177.092,6.194,148.253
C09882=1228.380,228.370,-58.904,-177.094,6.192,148.253
C09883=1228.385,228.122,-58.878,-177.097,6.190,148.254
C09884=1228.389,227.872,-58.853,-177.099,6.188,148.254
C09885=1228.394,227.624,-58.828,-177.102,6.186,148.254
C09886=1228.399,227.375,-58.803,-177.105,6.184,148.255
C09887=1228.404,227.127,-58.777,-177.107,6.182,148.255
C09888=1228.408,226.878,-58.752,-177.109,6.180,148.255
C09889=1228.413,226.629,-58.727,-177.112,6.178,148.256
C09890=1228.416,226.381,-58.702,-177.115,6.177,148.256
C09891=1228.421,226.132,-58.677,-177.117,6.176,148.256
C09892=1228.426,225.883,-58.651,-177.119,6.174,148.257
C09893=1228.430,225.634,-58.626,-177.122,6.172,148.257
C09894=1228.435,225.386,-58.601,-177.125,6.170,148.257
C09895=1228.439,225.137,-58.576,-177.127,6.168,148.258
C09896=1228.444,224.889,-58.551,-177.130,6.166,148.258
C09897=1228.448,224.640,-58.525,-177.133,6.164,148.258
C09898=1228.453,224.391,-58.501,-177.135,6.162,148.258
C09899=1228.457,224.142,-58.475,-177.138,6.161,148.259
C09900=1228.462,223.894,-58.451,-177.140,6.160,148.259
C09901=1228.466,223.644,-58.426,-177.142,6.158,148.260
C09902=1228.471,223.396,-58.400,-177.145,6.156,148.260
C09903=1228.476,223.148,-58.376,-177.148,6.154,148.260
C09904=1228.480,222.899,-58.351,-177.150,6.152,148.260
C09905=1228.485,222.650,-58.326,-177.153,6.150,148.261
C09906=1228.489,222.402,-58.300,-177.156,6.148,148.261
C09907=1228.494,222.153,-58.276,-177.158,6.146,148.261
C09908=1228.498,221.904,-58.251,-177.160,6.145,148.262
C09909=1228.503,221.656,-58.226,-177.163,6.144,148.262
C09910=1228.507,221.406,-58.201,-177.166,6.142,148.262
C09911=1228.511,221.158,-58.176,-177.168,6.140,148.263
C09912=1228.516,220.909,-58.151,-177.171,6.138,148.263
C09913=1228.521,220.660,-58.126,-177.173,6.136,148.263
C09914=1228.525,220.412,-58.101,-177.176,6.134,148.264
C09915=1228.530,220.163,-58.076,-177.179,6.132,148.264
C09916=1228.535,219.914,-58.052,-177.181,6.131,148.264
C09917=1228.539,219.665,-58.027,-177.183,6.129,148.265
C09918=1228.543,219.417,-58.002,-177.186,6.128,148.265
C09919=1228.548,219.168,-57.977,-177.189,6.126,148.265
C09920=1228.552,218.919,-57.953,-177.191,6.124,148.266
C09921=1228.557,218.670,-57.928,-177.194,6.122,148.266
C09922=1228.561,218.422,-57.903,-177.197,6.120,148.266
C09923=1228.566,218.173,-57.878,-177.199,6.119,148.267
C09924=1228.571,217.924,-57.853,-177.201,6.117,148.267
C09925=1228.575,217.675,-57.829,-177.204,6.115,148.267
C09926=1228.580,217.427,-57.804,-177.206,6.114,148.268
C09927=1228.584,217.178,-57.779,-177.209,6.112,148.268
C09928=1228.589,216.929,-57.755,-177.212,6.110,148.268
C09929=1228.593,216.681,-57.731,-177.214,6.108,148.269
C09930=1228.598,216.432,-57.706,-177.216,6.107,148.269
C09931=1228.603,216.183,-57.681,-177.219,6.105,148.269
C09932=1228.607,215.935,-57.656,-177.222,6.103,148.270
C09933=1228.611,215.686,-57.631,-177.224,6.101,148.270
C09934=1228.616,215.437,-57.607,-177.227,6.099,148.270
C09935=1228.621,215.189,-57.582,-177.230,6.098,148.271
C09936=1228.625,214.939,-57.558,-177.232,6.096,148.271
C09937=1228.630,214.691,-57.533,-177.234,6.095,148.271
C09938=1228.634,214.442,-57.509,-177.237,6.093,148.272
C09939=1228.639,214.193,-57.484,-177.240,6.091,148.272
C09940=1228.643,213.944,-57.460,-177.242,6.089,148.272
C09941=1228.648,213.696,-57.435,-177.245,6.087,148.273
C09942=1228.652,213.447,-57.411,-177.247,6.085,148.273
C09943=1228.657,213.198,-57.386,-177.250,6.084,148.274
C09944=1228.662,212.950,-57.362,-177.252,6.083,148.274
C09945=1228.665,212.700,-57.338,-177.255,6.081,148.274
C09946=1228.671,212.452,-57.313,-177.258,6.079,148.275
C09947=1228.675,212.203,-57.289,-177.261,6.077,148.275
C09948=1228.680,211.933,-57.262,-177.263,6.075,148.275
C09949=1228.685,211.662,-57.235,-177.266,6.074,148.276
C09950=1228.690,211.391,-57.209,-177.268,6.072,148.276
C09951=1228.695,211.121,-57.182,-177.272,6.070,148.277
C09952=1228.700,210.873,-57.158,-177.274,6.068,148.277
C09953=1228.703,210.624,-57.134,-177.277,6.066,148.277
C09954=1228.709,210.375,-57.109,-177.279,6.065,148.278
C09955=1228.713,210.127,-57.085,-177.281,6.064,148.278
C09956=1228.717,209.878,-57.061,-177.284,6.062,148.278
C09957=1228.722,209.629,-57.036,-177.287,6.060,148.279
C09958=1228.727,209.380,-57.013,-177.289,6.058,148.279
C09959=1228.732,209.131,-56.988,-177.292,6.056,148.279
C09960=1228.736,208.883,-56.964,-177.294,6.055,148.280
C09961=1228.741,208.634,-56.940,-177.297,6.053,148.280
C09962=1228.745,208.385,-56.915,-177.299,6.051,148.280
C09963=1228.750,208.136,-56.892,-177.302,6.050,148.281
C09964=1228.754,207.887,-56.867,-177.305,6.048,148.281
C09965=1228.759,207.639,-56.843,-177.307,6.047,148.282
C09966=1228.764,207.390,-56.819,-177.310,6.045,148.282
C09967=1228.767,207.141,-56.794,-177.312,6.043,148.282
C09968=1228.772,206.892,-56.771,-177.315,6.041,148.283
C09969=1228.777,206.643,-56.746,-177.318,6.040,148.283
C09970=1228.782,206.395,-56.722,-177.320,6.038,148.283
C09971=1228.786,206.146,-56.699,-177.322,6.037,148.284
C09972=1228.790,205.897,-56.674,-177.325,6.035,148.284
C09973=1228.795,205.648,-56.650,-177.328,6.033,148.284
C09974=1228.800,205.400,-56.626,-177.330,6.032,148.285
C09975=1228.804,205.151,-56.602,-177.333,6.030,148.285
C09976=1228.809,204.902,-56.578,-177.336,6.029,148.286
C09977=1228.814,204.653,-56.554,-177.338,6.027,148.286
C09978=1228.818,204.404,-56.530,-177.341,6.025,148.286
C09979=1228.822,204.155,-56.506,-177.343,6.024,148.287
C09980=1228.827,203.906,-56.482,-177.346,6.022,148.287
C09981=1228.832,203.658,-56.458,-177.348,6.020,148.287
C09982=1228.837,203.409,-56.434,-177.351,6.018,148.288
C09983=1228.841,203.160,-56.410,-177.353,6.017,148.288
C09984=1228.846,202.912,-56.386,-177.356,6.015,148.288
C09985=1228.850,202.663,-56.363,-177.359,6.014,148.289
C09986=1228.854,202.414,-56.338,-177.361,6.012,148.289
C09987=1228.859,202.165,-56.315,-177.363,6.011,148.290
C09988=1228.863,201.916,-56.291,-177.366,6.009,148.290
C09989=1228.869,201.667,-56.267,-177.369,6.007,148.290
C09990=1228.873,201.418,-56.243,-177.371,6.005,148.291
C09991=1228.878,201.170,-56.219,-177.373,6.004,148.291
C09992=1228.882,200.921,-56.195,-177.376,6.002,148.291
C09993=1228.887,200.672,-56.172,-177.379,6.001,148.292
C09994=1228.891,200.423,-56.148,-177.382,5.999,148.292
C09995=1228.896,200.174,-56.125,-177.384,5.998,148.293
C09996=1228.900,199.926,-56.101,-177.386,5.996,148.293
//INST
///DATE 2021/06/15 17:21
///ATTR SC,RW,RJ
////FRAME ROBOT
///GROUP1 RB1
NOP
MOVL C00000 V=800.0 PL=0
MOVL C00001 V=800.0 PL=0
MOVL C00002 V=800.0 PL=0
MOVL C00003 V=800.0 PL=0
MOVL C00004 V=800.0 PL=0
MOVL C00005 V=800.0 PL=0
MOVL C00006 V=800.0 PL=0
MOVL C00007 V=800.0 PL=0
MOVL C00008 V=800.0 PL=0
MOVL C00009 V=800.0 PL=0
MOVL C00010 V=800.0 PL=0
MOVL C00011 V=800.0 PL=0
MOVL C00012 V=800.0 PL=0
MOVL C00013 V=800.0 PL=0
MOVL C00014 V=800.0 PL=0
MOVL C00015 V=800.0 PL=0
MOVL C00016 V=800.0 PL=0
MOVL C00017 V=800.0 PL=0
MOVL C00018 V=800.0 PL=0
MOVL C00019 V=800.0 PL=0
MOVL C00020 V=800.0 PL=0
MOVL C00021 V=800.0 PL=0
MOVL C00022 V=800.0 PL=0
MOVL C00023 V=800.0 PL=0
MOVL C00024 V=800.0 PL=0
MOVL C00025 V=800.0 PL=0
MOVL C00026 V=800.0 PL=0
MOVL C00027 V=800.0 PL=0
MOVL C00028 V=800.0 PL=0
MOVL C00029 V=800.0 PL=0
MOVL C00030 V=800.0 PL=0
MOVL C00031 V=800.0 PL=0
MOVL C00032 V=800.0 PL=0
MOVL C00033 V=800.0 PL=0
MOVL C00034 V=800.0 PL=0
MOVL C00035 V=800.0 PL=0
MOVL C00036 V=800.0 PL=0
MOVL C00037 V=800.0 PL=0
MOVL C00038 V=800.0 PL=0
MOVL C00039 V=800.0 PL=0
MOVL C00040 V=800.0 PL=0
MOVL C00041 V=800.0 PL=0
MOVL C00042 V=800.0 PL=0
MOVL C00043 V=800.0 PL=0
MOVL C00044 V=800.0 PL=0
MOVL C00045 V=800.0 PL=0
MOVL C00046 V=800.0 PL=0
MOVL C00047 V=800.0 PL=0
MOVL C00048 V=800.0 PL=0
MOVL C00049 V=800.0 PL=0
MOVL C00050 V=800.0 PL=0
MOVL C00051 V=800.0 PL=0
MOVL C00052 V=800.0 PL=0
MOVL C00053 V=800.0 PL=0
MOVL C00054 V=800.0 PL=0
MOVL C00055 V=800.0 PL=0
MOVL C00056 V=800.0 PL=0
MOVL C00057 V=800.0 PL=0
MOVL C00058 V=800.0 PL=0
MOVL C00059 V=800.0 PL=0
MOVL C00060 V=800.0 PL=0
MOVL C00061 V=800.0 PL=0
MOVL C00062 V=800.0 PL=0
MOVL C00063 V=800.0 PL=0
MOVL C00064 V=800.0 PL=0
MOVL C00065 V=800.0 PL=0
MOVL C00066 V=800.0 PL=0
MOVL C00067 V=800.0 PL=0
MOVL C00068 V=800.0 PL=0
MOVL C00069 V=800.0 PL=0
MOVL C00070 V=800.0 PL=0
MOVL C00071 V=800.0 PL=0
MOVL C00072 V=800.0 PL=0
MOVL C00073 V=800.0 PL=0
MOVL C00074 V=800.0 PL=0
MOVL C00075 V=800.0 PL=0
MOVL C00076 V=800.0 PL=0
MOVL C00077 V=800.0 PL=0
MOVL C00078 V=800.0 PL=0
MOVL C00079 V=800.0 PL=0
MOVL C00080 V=800.0 PL=0
MOVL C00081 V=800.0 PL=0
MOVL C00082 V=800.0 PL=0
MOVL C00083 V=800.0 PL=0
MOVL C00084 V=800.0 PL=0
MOVL C00085 V=800.0 PL=0
MOVL C00086 V=800.0 PL=0
MOVL C00087 V=800.0 PL=0
MOVL C00088 V=800.0 PL=0
MOVL C00089 V=800.0 PL=0
MOVL C00090 V=800.0 PL=0
MOVL C00091 V=800.0 PL=0
MOVL C00092 V=800.0 PL=0
MOVL C00093 V=800.0 PL=0
MOVL C00094 V=800.0 PL=0
MOVL C00095 V=800.0 PL=0
MOVL C00096 V=800.0 PL=0
MOVL C00097 V=800.0 PL=0
MOVL C00098 V=800.0 PL=0
MOVL C00099 V=800.0 PL=0
MOVL C00100 V=800.0 PL=0
MOVL C00101 V=800.0 PL=0
MOVL C00102 V=800.0 PL=0
MOVL C00103 V=800.0 PL=0
MOVL C00104 V=800.0 PL=0
MOVL C00105 V=800.0 PL=0
MOVL C00106 V=800.0 PL=0
MOVL C00107 V=800.0 PL=0
MOVL C00108 V=800.0 PL=0
MOVL C00109 V=800.0 PL=0
MOVL C00110 V=800.0 PL=0
MOVL C00111 V=800.0 PL=0
MOVL C00112 V=800.0 PL=0
MOVL C00113 V=800.0 PL=0
MOVL C00114 V=800.0 PL=0
MOVL C00115 V=800.0 PL=0
MOVL C00116 V=800.0 PL=0
MOVL C00117 V=800.0 PL=0
MOVL C00118 V=800.0 PL=0
MOVL C00119 V=800.0 PL=0
MOVL C00120 V=800.0 PL=0
MOVL C00121 V=800.0 PL=0
MOVL C00122 V=800.0 PL=0
MOVL C00123 V=800.0 PL=0
MOVL C00124 V=800.0 PL=0
MOVL C00125 V=800.0 PL=0
MOVL C00126 V=800.0 PL=0
MOVL C00127 V=800.0 PL=0
MOVL C00128 V=800.0 PL=0
MOVL C00129 V=800.0 PL=0
MOVL C00130 V=800.0 PL=0
MOVL C00131 V=800.0 PL=0
MOVL C00132 V=800.0 PL=0
MOVL C00133 V=800.0 PL=0
MOVL C00134 V=800.0 PL=0
MOVL C00135 V=800.0 PL=0
MOVL C00136 V=800.0 PL=0
MOVL C00137 V=800.0 PL=0
MOVL C00138 V=800.0 PL=0
MOVL C00139 V=800.0 PL=0
MOVL C00140 V=800.0 PL=0
MOVL C00141 V=800.0 PL=0
MOVL C00142 V=800.0 PL=0
MOVL C00143 V=800.0 PL=0
MOVL C00144 V=800.0 PL=0
MOVL C00145 V=800.0 PL=0
MOVL C00146 V=800.0 PL=0
MOVL C00147 V=800.0 PL=0
MOVL C00148 V=800.0 PL=0
MOVL C00149 V=800.0 PL=0
MOVL C00150 V=800.0 PL=0
MOVL C00151 V=800.0 PL=0
MOVL C00152 V=800.0 PL=0
MOVL C00153 V=800.0 PL=0
MOVL C00154 V=800.0 PL=0
MOVL C00155 V=800.0 PL=0
MOVL C00156 V=800.0 PL=0
MOVL C00157 V=800.0 PL=0
MOVL C00158 V=800.0 PL=0
MOVL C00159 V=800.0 PL=0
MOVL C00160 V=800.0 PL=0
MOVL C00161 V=800.0 PL=0
MOVL C00162 V=800.0 PL=0
MOVL C00163 V=800.0 PL=0
MOVL C00164 V=800.0 PL=0
MOVL C00165 V=800.0 PL=0
MOVL C00166 V=800.0 PL=0
MOVL C00167 V=800.0 PL=0
MOVL C00168 V=800.0 PL=0
MOVL C00169 V=800.0 PL=0
MOVL C00170 V=800.0 PL=0
MOVL C00171 V=800.0 PL=0
MOVL C00172 V=800.0 PL=0
MOVL C00173 V=800.0 PL=0
MOVL C00174 V=800.0 PL=0
MOVL C00175 V=800.0 PL=0
MOVL C00176 V=800.0 PL=0
MOVL C00177 V=800.0 PL=0
MOVL C00178 V=800.0 PL=0
MOVL C00179 V=800.0 PL=0
MOVL C00180 V=800.0 PL=0
MOVL C00181 V=800.0 PL=0
MOVL C00182 V=800.0 PL=0
MOVL C00183 V=800.0 PL=0
MOVL C00184 V=800.0 PL=0
MOVL C00185 V=800.0 PL=0
MOVL C00186 V=800.0 PL=0
MOVL C00187 V=800.0 PL=0
MOVL C00188 V=800.0 PL=0
MOVL C00189 V=800.0 PL=0
MOVL C00190 V=800.0 PL=0
MOVL C00191 V=800.0 PL=0
MOVL C00192 V=800.0 PL=0
MOVL C00193 V=800.0 PL=0
MOVL C00194 V=800.0 PL=0
MOVL C00195 V=800.0 PL=0
MOVL C00196 V=800.0 PL=0
MOVL C00197 V=800.0 PL=0
MOVL C00198 V=800.0 PL=0
MOVL C00199 V=800.0 PL=0
MOVL C00200 V=800.0 PL=0
MOVL C00201 V=800.0 PL=0
MOVL C00202 V=800.0 PL=0
MOVL C00203 V=800.0 PL=0
MOVL C00204 V=800.0 PL=0
MOVL C00205 V=800.0 PL=0
MOVL C00206 V=800.0 PL=0
MOVL C00207 V=800.0 PL=0
MOVL C00208 V=800.0 PL=0
MOVL C00209 V=800.0 PL=0
MOVL C00210 V=800.0 PL=0
MOVL C00211 V=800.0 PL=0
MOVL C00212 V=800.0 PL=0
MOVL C00213 V=800.0 PL=0
MOVL C00214 V=800.0 PL=0
MOVL C00215 V=800.0 PL=0
MOVL C00216 V=800.0 PL=0
MOVL C00217 V=800.0 PL=0
MOVL C00218 V=800.0 PL=0
MOVL C00219 V=800.0 PL=0
MOVL C00220 V=800.0 PL=0
MOVL C00221 V=800.0 PL=0
MOVL C00222 V=800.0 PL=0
MOVL C00223 V=800.0 PL=0
MOVL C00224 V=800.0 PL=0
MOVL C00225 V=800.0 PL=0
MOVL C00226 V=800.0 PL=0
MOVL C00227 V=800.0 PL=0
MOVL C00228 V=800.0 PL=0
MOVL C00229 V=800.0 PL=0
MOVL C00230 V=800.0 PL=0
MOVL C00231 V=800.0 PL=0
MOVL C00232 V=800.0 PL=0
MOVL C00233 V=800.0 PL=0
MOVL C00234 V=800.0 PL=0
MOVL C00235 V=800.0 PL=0
MOVL C00236 V=800.0 PL=0
MOVL C00237 V=800.0 PL=0
MOVL C00238 V=800.0 PL=0
MOVL C00239 V=800.0 PL=0
MOVL C00240 V=800.0 PL=0
MOVL C00241 V=800.0 PL=0
MOVL C00242 V=800.0 PL=0
MOVL C00243 V=800.0 PL=0
MOVL C00244 V=800.0 PL=0
MOVL C00245 V=800.0 PL=0
MOVL C00246 V=800.0 PL=0
MOVL C00247 V=800.0 PL=0
MOVL C00248 V=800.0 PL=0
MOVL C00249 V=800.0 PL=0
MOVL C00250 V=800.0 PL=0
MOVL C00251 V=800.0 PL=0
MOVL C00252 V=800.0 PL=0
MOVL C00253 V=800.0 PL=0
MOVL C00254 V=800.0 PL=0
MOVL C00255 V=800.0 PL=0
MOVL C00256 V=800.0 PL=0
MOVL C00257 V=800.0 PL=0
MOVL C00258 V=800.0 PL=0
MOVL C00259 V=800.0 PL=0
MOVL C00260 V=800.0 PL=0
MOVL C00261 V=800.0 PL=0
MOVL C00262 V=800.0 PL=0
MOVL C00263 V=800.0 PL=0
MOVL C00264 V=800.0 PL=0
MOVL C00265 V=800.0 PL=0
MOVL C00266 V=800.0 PL=0
MOVL C00267 V=800.0 PL=0
MOVL C00268 V=800.0 PL=0
MOVL C00269 V=800.0 PL=0
MOVL C00270 V=800.0 PL=0
MOVL C00271 V=800.0 PL=0
MOVL C00272 V=800.0 PL=0
MOVL C00273 V=800.0 PL=0
MOVL C00274 V=800.0 PL=0
MOVL C00275 V=800.0 PL=0
MOVL C00276 V=800.0 PL=0
MOVL C00277 V=800.0 PL=0
MOVL C00278 V=800.0 PL=0
MOVL C00279 V=800.0 PL=0
MOVL C00280 V=800.0 PL=0
MOVL C00281 V=800.0 PL=0
MOVL C00282 V=800.0 PL=0
MOVL C00283 V=800.0 PL=0
MOVL C00284 V=800.0 PL=0
MOVL C00285 V=800.0 PL=0
MOVL C00286 V=800.0 PL=0
MOVL C00287 V=800.0 PL=0
MOVL C00288 V=800.0 PL=0
MOVL C00289 V=800.0 PL=0
MOVL C00290 V=800.0 PL=0
MOVL C00291 V=800.0 PL=0
MOVL C00292 V=800.0 PL=0
MOVL C00293 V=800.0 PL=0
MOVL C00294 V=800.0 PL=0
MOVL C00295 V=800.0 PL=0
MOVL C00296 V=800.0 PL=0
MOVL C00297 V=800.0 PL=0
MOVL C00298 V=800.0 PL=0
MOVL C00299 V=800.0 PL=0
MOVL C00300 V=800.0 PL=0
MOVL C00301 V=800.0 PL=0
MOVL C00302 V=800.0 PL=0
MOVL C00303 V=800.0 PL=0
MOVL C00304 V=800.0 PL=0
MOVL C00305 V=800.0 PL=0
MOVL C00306 V=800.0 PL=0
MOVL C00307 V=800.0 PL=0
MOVL C00308 V=800.0 PL=0
MOVL C00309 V=800.0 PL=0
MOVL C00310 V=800.0 PL=0
MOVL C00311 V=800.0 PL=0
MOVL C00312 V=800.0 PL=0
MOVL C00313 V=800.0 PL=0
MOVL C00314 V=800.0 PL=0
MOVL C00315 V=800.0 PL=0
MOVL C00316 V=800.0 PL=0
MOVL C00317 V=800.0 PL=0
MOVL C00318 V=800.0 PL=0
MOVL C00319 V=800.0 PL=0
MOVL C00320 V=800.0 PL=0
MOVL C00321 V=800.0 PL=0
MOVL C00322 V=800.0 PL=0
MOVL C00323 V=800.0 PL=0
MOVL C00324 V=800.0 PL=0
MOVL C00325 V=800.0 PL=0
MOVL C00326 V=800.0 PL=0
MOVL C00327 V=800.0 PL=0
MOVL C00328 V=800.0 PL=0
MOVL C00329 V=800.0 PL=0
MOVL C00330 V=800.0 PL=0
MOVL C00331 V=800.0 PL=0
MOVL C00332 V=800.0 PL=0
MOVL C00333 V=800.0 PL=0
MOVL C00334 V=800.0 PL=0
MOVL C00335 V=800.0 PL=0
MOVL C00336 V=800.0 PL=0
MOVL C00337 V=800.0 PL=0
MOVL C00338 V=800.0 PL=0
MOVL C00339 V=800.0 PL=0
MOVL C00340 V=800.0 PL=0
MOVL C00341 V=800.0 PL=0
MOVL C00342 V=800.0 PL=0
MOVL C00343 V=800.0 PL=0
MOVL C00344 V=800.0 PL=0
MOVL C00345 V=800.0 PL=0
MOVL C00346 V=800.0 PL=0
MOVL C00347 V=800.0 PL=0
MOVL C00348 V=800.0 PL=0
MOVL C00349 V=800.0 PL=0
MOVL C00350 V=800.0 PL=0
MOVL C00351 V=800.0 PL=0
MOVL C00352 V=800.0 PL=0
MOVL C00353 V=800.0 PL=0
MOVL C00354 V=800.0 PL=0
MOVL C00355 V=800.0 PL=0
MOVL C00356 V=800.0 PL=0
MOVL C00357 V=800.0 PL=0
MOVL C00358 V=800.0 PL=0
MOVL C00359 V=800.0 PL=0
MOVL C00360 V=800.0 PL=0
MOVL C00361 V=800.0 PL=0
MOVL C00362 V=800.0 PL=0
MOVL C00363 V=800.0 PL=0
MOVL C00364 V=800.0 PL=0
MOVL C00365 V=800.0 PL=0
MOVL C00366 V=800.0 PL=0
MOVL C00367 V=800.0 PL=0
MOVL C00368 V=800.0 PL=0
MOVL C00369 V=800.0 PL=0
MOVL C00370 V=800.0 PL=0
MOVL C00371 V=800.0 PL=0
MOVL C00372 V=800.0 PL=0
MOVL C00373 V=800.0 PL=0
MOVL C00374 V=800.0 PL=0
MOVL C00375 V=800.0 PL=0
MOVL C00376 V=800.0 PL=0
MOVL C00377 V=800.0 PL=0
MOVL C00378 V=800.0 PL=0
MOVL C00379 V=800.0 PL=0
MOVL C00380 V=800.0 PL=0
MOVL C00381 V=800.0 PL=0
MOVL C00382 V=800.0 PL=0
MOVL C00383 V=800.0 PL=0
MOVL C00384 V=800.0 PL=0
MOVL C00385 V=800.0 PL=0
MOVL C00386 V=800.0 PL=0
MOVL C00387 V=800.0 PL=0
MOVL C00388 V=800.0 PL=0
MOVL C00389 V=800.0 PL=0
MOVL C00390 V=800.0 PL=0
MOVL C00391 V=800.0 PL=0
MOVL C00392 V=800.0 PL=0
MOVL C00393 V=800.0 PL=0
MOVL C00394 V=800.0 PL=0
MOVL C00395 V=800.0 PL=0
MOVL C00396 V=800.0 PL=0
MOVL C00397 V=800.0 PL=0
MOVL C00398 V=800.0 PL=0
MOVL C00399 V=800.0 PL=0
MOVL C00400 V=800.0 PL=0
MOVL C00401 V=800.0 PL=0
MOVL C00402 V=800.0 PL=0
MOVL C00403 V=800.0 PL=0
MOVL C00404 V=800.0 PL=0
MOVL C00405 V=800.0 PL=0
MOVL C00406 V=800.0 PL=0
MOVL C00407 V=800.0 PL=0
MOVL C00408 V=800.0 PL=0
MOVL C00409 V=800.0 PL=0
MOVL C00410 V=800.0 PL=0
MOVL C00411 V=800.0 PL=0
MOVL C00412 V=800.0 PL=0
MOVL C00413 V=800.0 PL=0
MOVL C00414 V=800.0 PL=0
MOVL C00415 V=800.0 PL=0
MOVL C00416 V=800.0 PL=0
MOVL C00417 V=800.0 PL=0
MOVL C00418 V=800.0 PL=0
MOVL C00419 V=800.0 PL=0
MOVL C00420 V=800.0 PL=0
MOVL C00421 V=800.0 PL=0
MOVL C00422 V=800.0 PL=0
MOVL C00423 V=800.0 PL=0
MOVL C00424 V=800.0 PL=0
MOVL C00425 V=800.0 PL=0
MOVL C00426 V=800.0 PL=0
MOVL C00427 V=800.0 PL=0
MOVL C00428 V=800.0 PL=0
MOVL C00429 V=800.0 PL=0
MOVL C00430 V=800.0 PL=0
MOVL C00431 V=800.0 PL=0
MOVL C00432 V=800.0 PL=0
MOVL C00433 V=800.0 PL=0
MOVL C00434 V=800.0 PL=0
MOVL C00435 V=800.0 PL=0
MOVL C00436 V=800.0 PL=0
MOVL C00437 V=800.0 PL=0
MOVL C00438 V=800.0 PL=0
MOVL C00439 V=800.0 PL=0
MOVL C00440 V=800.0 PL=0
MOVL C00441 V=800.0 PL=0
MOVL C00442 V=800.0 PL=0
MOVL C00443 V=800.0 PL=0
MOVL C00444 V=800.0 PL=0
MOVL C00445 V=800.0 PL=0
MOVL C00446 V=800.0 PL=0
MOVL C00447 V=800.0 PL=0
MOVL C00448 V=800.0 PL=0
MOVL C00449 V=800.0 PL=0
MOVL C00450 V=800.0 PL=0
MOVL C00451 V=800.0 PL=0
MOVL C00452 V=800.0 PL=0
MOVL C00453 V=800.0 PL=0
MOVL C00454 V=800.0 PL=0
MOVL C00455 V=800.0 PL=0
MOVL C00456 V=800.0 PL=0
MOVL C00457 V=800.0 PL=0
MOVL C00458 V=800.0 PL=0
MOVL C00459 V=800.0 PL=0
MOVL C00460 V=800.0 PL=0
MOVL C00461 V=800.0 PL=0
MOVL C00462 V=800.0 PL=0
MOVL C00463 V=800.0 PL=0
MOVL C00464 V=800.0 PL=0
MOVL C00465 V=800.0 PL=0
MOVL C00466 V=800.0 PL=0
MOVL C00467 V=800.0 PL=0
MOVL C00468 V=800.0 PL=0
MOVL C00469 V=800.0 PL=0
MOVL C00470 V=800.0 PL=0
MOVL C00471 V=800.0 PL=0
MOVL C00472 V=800.0 PL=0
MOVL C00473 V=800.0 PL=0
MOVL C00474 V=800.0 PL=0
MOVL C00475 V=800.0 PL=0
MOVL C00476 V=800.0 PL=0
MOVL C00477 V=800.0 PL=0
MOVL C00478 V=800.0 PL=0
MOVL C00479 V=800.0 PL=0
MOVL C00480 V=800.0 PL=0
MOVL C00481 V=800.0 PL=0
MOVL C00482 V=800.0 PL=0
MOVL C00483 V=800.0 PL=0
MOVL C00484 V=800.0 PL=0
MOVL C00485 V=800.0 PL=0
MOVL C00486 V=800.0 PL=0
MOVL C00487 V=800.0 PL=0
MOVL C00488 V=800.0 PL=0
MOVL C00489 V=800.0 PL=0
MOVL C00490 V=800.0 PL=0
MOVL C00491 V=800.0 PL=0
MOVL C00492 V=800.0 PL=0
MOVL C00493 V=800.0 PL=0
MOVL C00494 V=800.0 PL=0
MOVL C00495 V=800.0 PL=0
MOVL C00496 V=800.0 PL=0
MOVL C00497 V=800.0 PL=0
MOVL C00498 V=800.0 PL=0
MOVL C00499 V=800.0 PL=0
MOVL C00500 V=800.0 PL=0
MOVL C00501 V=800.0 PL=0
MOVL C00502 V=800.0 PL=0
MOVL C00503 V=800.0 PL=0
MOVL C00504 V=800.0 PL=0
MOVL C00505 V=800.0 PL=0
MOVL C00506 V=800.0 PL=0
MOVL C00507 V=800.0 PL=0
MOVL C00508 V=800.0 PL=0
MOVL C00509 V=800.0 PL=0
MOVL C00510 V=800.0 PL=0
MOVL C00511 V=800.0 PL=0
MOVL C00512 V=800.0 PL=0
MOVL C00513 V=800.0 PL=0
MOVL C00514 V=800.0 PL=0
MOVL C00515 V=800.0 PL=0
MOVL C00516 V=800.0 PL=0
MOVL C00517 V=800.0 PL=0
MOVL C00518 V=800.0 PL=0
MOVL C00519 V=800.0 PL=0
MOVL C00520 V=800.0 PL=0
MOVL C00521 V=800.0 PL=0
MOVL C00522 V=800.0 PL=0
MOVL C00523 V=800.0 PL=0
MOVL C00524 V=800.0 PL=0
MOVL C00525 V=800.0 PL=0
MOVL C00526 V=800.0 PL=0
MOVL C00527 V=800.0 PL=0
MOVL C00528 V=800.0 PL=0
MOVL C00529 V=800.0 PL=0
MOVL C00530 V=800.0 PL=0
MOVL C00531 V=800.0 PL=0
MOVL C00532 V=800.0 PL=0
MOVL C00533 V=800.0 PL=0
MOVL C00534 V=800.0 PL=0
MOVL C00535 V=800.0 PL=0
MOVL C00536 V=800.0 PL=0
MOVL C00537 V=800.0 PL=0
MOVL C00538 V=800.0 PL=0
MOVL C00539 V=800.0 PL=0
MOVL C00540 V=800.0 PL=0
MOVL C00541 V=800.0 PL=0
MOVL C00542 V=800.0 PL=0
MOVL C00543 V=800.0 PL=0
MOVL C00544 V=800.0 PL=0
MOVL C00545 V=800.0 PL=0
MOVL C00546 V=800.0 PL=0
MOVL C00547 V=800.0 PL=0
MOVL C00548 V=800.0 PL=0
MOVL C00549 V=800.0 PL=0
MOVL C00550 V=800.0 PL=0
MOVL C00551 V=800.0 PL=0
MOVL C00552 V=800.0 PL=0
MOVL C00553 V=800.0 PL=0
MOVL C00554 V=800.0 PL=0
MOVL C00555 V=800.0 PL=0
MOVL C00556 V=800.0 PL=0
MOVL C00557 V=800.0 PL=0
MOVL C00558 V=800.0 PL=0
MOVL C00559 V=800.0 PL=0
MOVL C00560 V=800.0 PL=0
MOVL C00561 V=800.0 PL=0
MOVL C00562 V=800.0 PL=0
MOVL C00563 V=800.0 PL=0
MOVL C00564 V=800.0 PL=0
MOVL C00565 V=800.0 PL=0
MOVL C00566 V=800.0 PL=0
MOVL C00567 V=800.0 PL=0
MOVL C00568 V=800.0 PL=0
MOVL C00569 V=800.0 PL=0
MOVL C00570 V=800.0 PL=0
MOVL C00571 V=800.0 PL=0
MOVL C00572 V=800.0 PL=0
MOVL C00573 V=800.0 PL=0
MOVL C00574 V=800.0 PL=0
MOVL C00575 V=800.0 PL=0
MOVL C00576 V=800.0 PL=0
MOVL C00577 V=800.0 PL=0
MOVL C00578 V=800.0 PL=0
MOVL C00579 V=800.0 PL=0
MOVL C00580 V=800.0 PL=0
MOVL C00581 V=800.0 PL=0
MOVL C00582 V=800.0 PL=0
MOVL C00583 V=800.0 PL=0
MOVL C00584 V=800.0 PL=0
MOVL C00585 V=800.0 PL=0
MOVL C00586 V=800.0 PL=0
MOVL C00587 V=800.0 PL=0
MOVL C00588 V=800.0 PL=0
MOVL C00589 V=800.0 PL=0
MOVL C00590 V=800.0 PL=0
MOVL C00591 V=800.0 PL=0
MOVL C00592 V=800.0 PL=0
MOVL C00593 V=800.0 PL=0
MOVL C00594 V=800.0 PL=0
MOVL C00595 V=800.0 PL=0
MOVL C00596 V=800.0 PL=0
MOVL C00597 V=800.0 PL=0
MOVL C00598 V=800.0 PL=0
MOVL C00599 V=800.0 PL=0
MOVL C00600 V=800.0 PL=0
MOVL C00601 V=800.0 PL=0
MOVL C00602 V=800.0 PL=0
MOVL C00603 V=800.0 PL=0
MOVL C00604 V=800.0 PL=0
MOVL C00605 V=800.0 PL=0
MOVL C00606 V=800.0 PL=0
MOVL C00607 V=800.0 PL=0
MOVL C00608 V=800.0 PL=0
MOVL C00609 V=800.0 PL=0
MOVL C00610 V=800.0 PL=0
MOVL C00611 V=800.0 PL=0
MOVL C00612 V=800.0 PL=0
MOVL C00613 V=800.0 PL=0
MOVL C00614 V=800.0 PL=0
MOVL C00615 V=800.0 PL=0
MOVL C00616 V=800.0 PL=0
MOVL C00617 V=800.0 PL=0
MOVL C00618 V=800.0 PL=0
MOVL C00619 V=800.0 PL=0
MOVL C00620 V=800.0 PL=0
MOVL C00621 V=800.0 PL=0
MOVL C00622 V=800.0 PL=0
MOVL C00623 V=800.0 PL=0
MOVL C00624 V=800.0 PL=0
MOVL C00625 V=800.0 PL=0
MOVL C00626 V=800.0 PL=0
MOVL C00627 V=800.0 PL=0
MOVL C00628 V=800.0 PL=0
MOVL C00629 V=800.0 PL=0
MOVL C00630 V=800.0 PL=0
MOVL C00631 V=800.0 PL=0
MOVL C00632 V=800.0 PL=0
MOVL C00633 V=800.0 PL=0
MOVL C00634 V=800.0 PL=0
MOVL C00635 V=800.0 PL=0
MOVL C00636 V=800.0 PL=0
MOVL C00637 V=800.0 PL=0
MOVL C00638 V=800.0 PL=0
MOVL C00639 V=800.0 PL=0
MOVL C00640 V=800.0 PL=0
MOVL C00641 V=800.0 PL=0
MOVL C00642 V=800.0 PL=0
MOVL C00643 V=800.0 PL=0
MOVL C00644 V=800.0 PL=0
MOVL C00645 V=800.0 PL=0
MOVL C00646 V=800.0 PL=0
MOVL C00647 V=800.0 PL=0
MOVL C00648 V=800.0 PL=0
MOVL C00649 V=800.0 PL=0
MOVL C00650 V=800.0 PL=0
MOVL C00651 V=800.0 PL=0
MOVL C00652 V=800.0 PL=0
MOVL C00653 V=800.0 PL=0
MOVL C00654 V=800.0 PL=0
MOVL C00655 V=800.0 PL=0
MOVL C00656 V=800.0 PL=0
MOVL C00657 V=800.0 PL=0
MOVL C00658 V=800.0 PL=0
MOVL C00659 V=800.0 PL=0
MOVL C00660 V=800.0 PL=0
MOVL C00661 V=800.0 PL=0
MOVL C00662 V=800.0 PL=0
MOVL C00663 V=800.0 PL=0
MOVL C00664 V=800.0 PL=0
MOVL C00665 V=800.0 PL=0
MOVL C00666 V=800.0 PL=0
MOVL C00667 V=800.0 PL=0
MOVL C00668 V=800.0 PL=0
MOVL C00669 V=800.0 PL=0
MOVL C00670 V=800.0 PL=0
MOVL C00671 V=800.0 PL=0
MOVL C00672 V=800.0 PL=0
MOVL C00673 V=800.0 PL=0
MOVL C00674 V=800.0 PL=0
MOVL C00675 V=800.0 PL=0
MOVL C00676 V=800.0 PL=0
MOVL C00677 V=800.0 PL=0
MOVL C00678 V=800.0 PL=0
MOVL C00679 V=800.0 PL=0
MOVL C00680 V=800.0 PL=0
MOVL C00681 V=800.0 PL=0
MOVL C00682 V=800.0 PL=0
MOVL C00683 V=800.0 PL=0
MOVL C00684 V=800.0 PL=0
MOVL C00685 V=800.0 PL=0
MOVL C00686 V=800.0 PL=0
MOVL C00687 V=800.0 PL=0
MOVL C00688 V=800.0 PL=0
MOVL C00689 V=800.0 PL=0
MOVL C00690 V=800.0 PL=0
MOVL C00691 V=800.0 PL=0
MOVL C00692 V=800.0 PL=0
MOVL C00693 V=800.0 PL=0
MOVL C00694 V=800.0 PL=0
MOVL C00695 V=800.0 PL=0
MOVL C00696 V=800.0 PL=0
MOVL C00697 V=800.0 PL=0
MOVL C00698 V=800.0 PL=0
MOVL C00699 V=800.0 PL=0
MOVL C00700 V=800.0 PL=0
MOVL C00701 V=800.0 PL=0
MOVL C00702 V=800.0 PL=0
MOVL C00703 V=800.0 PL=0
MOVL C00704 V=800.0 PL=0
MOVL C00705 V=800.0 PL=0
MOVL C00706 V=800.0 PL=0
MOVL C00707 V=800.0 PL=0
MOVL C00708 V=800.0 PL=0
MOVL C00709 V=800.0 PL=0
MOVL C00710 V=800.0 PL=0
MOVL C00711 V=800.0 PL=0
MOVL C00712 V=800.0 PL=0
MOVL C00713 V=800.0 PL=0
MOVL C00714 V=800.0 PL=0
MOVL C00715 V=800.0 PL=0
MOVL C00716 V=800.0 PL=0
MOVL C00717 V=800.0 PL=0
MOVL C00718 V=800.0 PL=0
MOVL C00719 V=800.0 PL=0
MOVL C00720 V=800.0 PL=0
MOVL C00721 V=800.0 PL=0
MOVL C00722 V=800.0 PL=0
MOVL C00723 V=800.0 PL=0
MOVL C00724 V=800.0 PL=0
MOVL C00725 V=800.0 PL=0
MOVL C00726 V=800.0 PL=0
MOVL C00727 V=800.0 PL=0
MOVL C00728 V=800.0 PL=0
MOVL C00729 V=800.0 PL=0
MOVL C00730 V=800.0 PL=0
MOVL C00731 V=800.0 PL=0
MOVL C00732 V=800.0 PL=0
MOVL C00733 V=800.0 PL=0
MOVL C00734 V=800.0 PL=0
MOVL C00735 V=800.0 PL=0
MOVL C00736 V=800.0 PL=0
MOVL C00737 V=800.0 PL=0
MOVL C00738 V=800.0 PL=0
MOVL C00739 V=800.0 PL=0
MOVL C00740 V=800.0 PL=0
MOVL C00741 V=800.0 PL=0
MOVL C00742 V=800.0 PL=0
MOVL C00743 V=800.0 PL=0
MOVL C00744 V=800.0 PL=0
MOVL C00745 V=800.0 PL=0
MOVL C00746 V=800.0 PL=0
MOVL C00747 V=800.0 PL=0
MOVL C00748 V=800.0 PL=0
MOVL C00749 V=800.0 PL=0
MOVL C00750 V=800.0 PL=0
MOVL C00751 V=800.0 PL=0
MOVL C00752 V=800.0 PL=0
MOVL C00753 V=800.0 PL=0
MOVL C00754 V=800.0 PL=0
MOVL C00755 V=800.0 PL=0
MOVL C00756 V=800.0 PL=0
MOVL C00757 V=800.0 PL=0
MOVL C00758 V=800.0 PL=0
MOVL C00759 V=800.0 PL=0
MOVL C00760 V=800.0 PL=0
MOVL C00761 V=800.0 PL=0
MOVL C00762 V=800.0 PL=0
MOVL C00763 V=800.0 PL=0
MOVL C00764 V=800.0 PL=0
MOVL C00765 V=800.0 PL=0
MOVL C00766 V=800.0 PL=0
MOVL C00767 V=800.0 PL=0
MOVL C00768 V=800.0 PL=0
MOVL C00769 V=800.0 PL=0
MOVL C00770 V=800.0 PL=0
MOVL C00771 V=800.0 PL=0
MOVL C00772 V=800.0 PL=0
MOVL C00773 V=800.0 PL=0
MOVL C00774 V=800.0 PL=0
MOVL C00775 V=800.0 PL=0
MOVL C00776 V=800.0 PL=0
MOVL C00777 V=800.0 PL=0
MOVL C00778 V=800.0 PL=0
MOVL C00779 V=800.0 PL=0
MOVL C00780 V=800.0 PL=0
MOVL C00781 V=800.0 PL=0
MOVL C00782 V=800.0 PL=0
MOVL C00783 V=800.0 PL=0
MOVL C00784 V=800.0 PL=0
MOVL C00785 V=800.0 PL=0
MOVL C00786 V=800.0 PL=0
MOVL C00787 V=800.0 PL=0
MOVL C00788 V=800.0 PL=0
MOVL C00789 V=800.0 PL=0
MOVL C00790 V=800.0 PL=0
MOVL C00791 V=800.0 PL=0
MOVL C00792 V=800.0 PL=0
MOVL C00793 V=800.0 PL=0
MOVL C00794 V=800.0 PL=0
MOVL C00795 V=800.0 PL=0
MOVL C00796 V=800.0 PL=0
MOVL C00797 V=800.0 PL=0
MOVL C00798 V=800.0 PL=0
MOVL C00799 V=800.0 PL=0
MOVL C00800 V=800.0 PL=0
MOVL C00801 V=800.0 PL=0
MOVL C00802 V=800.0 PL=0
MOVL C00803 V=800.0 PL=0
MOVL C00804 V=800.0 PL=0
MOVL C00805 V=800.0 PL=0
MOVL C00806 V=800.0 PL=0
MOVL C00807 V=800.0 PL=0
MOVL C00808 V=800.0 PL=0
MOVL C00809 V=800.0 PL=0
MOVL C00810 V=800.0 PL=0
MOVL C00811 V=800.0 PL=0
MOVL C00812 V=800.0 PL=0
MOVL C00813 V=800.0 PL=0
MOVL C00814 V=800.0 PL=0
MOVL C00815 V=800.0 PL=0
MOVL C00816 V=800.0 PL=0
MOVL C00817 V=800.0 PL=0
MOVL C00818 V=800.0 PL=0
MOVL C00819 V=800.0 PL=0
MOVL C00820 V=800.0 PL=0
MOVL C00821 V=800.0 PL=0
MOVL C00822 V=800.0 PL=0
MOVL C00823 V=800.0 PL=0
MOVL C00824 V=800.0 PL=0
MOVL C00825 V=800.0 PL=0
MOVL C00826 V=800.0 PL=0
MOVL C00827 V=800.0 PL=0
MOVL C00828 V=800.0 PL=0
MOVL C00829 V=800.0 PL=0
MOVL C00830 V=800.0 PL=0
MOVL C00831 V=800.0 PL=0
MOVL C00832 V=800.0 PL=0
MOVL C00833 V=800.0 PL=0
MOVL C00834 V=800.0 PL=0
MOVL C00835 V=800.0 PL=0
MOVL C00836 V=800.0 PL=0
MOVL C00837 V=800.0 PL=0
MOVL C00838 V=800.0 PL=0
MOVL C00839 V=800.0 PL=0
MOVL C00840 V=800.0 PL=0
MOVL C00841 V=800.0 PL=0
MOVL C00842 V=800.0 PL=0
MOVL C00843 V=800.0 PL=0
MOVL C00844 V=800.0 PL=0
MOVL C00845 V=800.0 PL=0
MOVL C00846 V=800.0 PL=0
MOVL C00847 V=800.0 PL=0
MOVL C00848 V=800.0 PL=0
MOVL C00849 V=800.0 PL=0
MOVL C00850 V=800.0 PL=0
MOVL C00851 V=800.0 PL=0
MOVL C00852 V=800.0 PL=0
MOVL C00853 V=800.0 PL=0
MOVL C00854 V=800.0 PL=0
MOVL C00855 V=800.0 PL=0
MOVL C00856 V=800.0 PL=0
MOVL C00857 V=800.0 PL=0
MOVL C00858 V=800.0 PL=0
MOVL C00859 V=800.0 PL=0
MOVL C00860 V=800.0 PL=0
MOVL C00861 V=800.0 PL=0
MOVL C00862 V=800.0 PL=0
MOVL C00863 V=800.0 PL=0
MOVL C00864 V=800.0 PL=0
MOVL C00865 V=800.0 PL=0
MOVL C00866 V=800.0 PL=0
MOVL C00867 V=800.0 PL=0
MOVL C00868 V=800.0 PL=0
MOVL C00869 V=800.0 PL=0
MOVL C00870 V=800.0 PL=0
MOVL C00871 V=800.0 PL=0
MOVL C00872 V=800.0 PL=0
MOVL C00873 V=800.0 PL=0
MOVL C00874 V=800.0 PL=0
MOVL C00875 V=800.0 PL=0
MOVL C00876 V=800.0 PL=0
MOVL C00877 V=800.0 PL=0
MOVL C00878 V=800.0 PL=0
MOVL C00879 V=800.0 PL=0
MOVL C00880 V=800.0 PL=0
MOVL C00881 V=800.0 PL=0
MOVL C00882 V=800.0 PL=0
MOVL C00883 V=800.0 PL=0
MOVL C00884 V=800.0 PL=0
MOVL C00885 V=800.0 PL=0
MOVL C00886 V=800.0 PL=0
MOVL C00887 V=800.0 PL=0
MOVL C00888 V=800.0 PL=0
MOVL C00889 V=800.0 PL=0
MOVL C00890 V=800.0 PL=0
MOVL C00891 V=800.0 PL=0
MOVL C00892 V=800.0 PL=0
MOVL C00893 V=800.0 PL=0
MOVL C00894 V=800.0 PL=0
MOVL C00895 V=800.0 PL=0
MOVL C00896 V=800.0 PL=0
MOVL C00897 V=800.0 PL=0
MOVL C00898 V=800.0 PL=0
MOVL C00899 V=800.0 PL=0
MOVL C00900 V=800.0 PL=0
MOVL C00901 V=800.0 PL=0
MOVL C00902 V=800.0 PL=0
MOVL C00903 V=800.0 PL=0
MOVL C00904 V=800.0 PL=0
MOVL C00905 V=800.0 PL=0
MOVL C00906 V=800.0 PL=0
MOVL C00907 V=800.0 PL=0
MOVL C00908 V=800.0 PL=0
MOVL C00909 V=800.0 PL=0
MOVL C00910 V=800.0 PL=0
MOVL C00911 V=800.0 PL=0
MOVL C00912 V=800.0 PL=0
MOVL C00913 V=800.0 PL=0
MOVL C00914 V=800.0 PL=0
MOVL C00915 V=800.0 PL=0
MOVL C00916 V=800.0 PL=0
MOVL C00917 V=800.0 PL=0
MOVL C00918 V=800.0 PL=0
MOVL C00919 V=800.0 PL=0
MOVL C00920 V=800.0 PL=0
MOVL C00921 V=800.0 PL=0
MOVL C00922 V=800.0 PL=0
MOVL C00923 V=800.0 PL=0
MOVL C00924 V=800.0 PL=0
MOVL C00925 V=800.0 PL=0
MOVL C00926 V=800.0 PL=0
MOVL C00927 V=800.0 PL=0
MOVL C00928 V=800.0 PL=0
MOVL C00929 V=800.0 PL=0
MOVL C00930 V=800.0 PL=0
MOVL C00931 V=800.0 PL=0
MOVL C00932 V=800.0 PL=0
MOVL C00933 V=800.0 PL=0
MOVL C00934 V=800.0 PL=0
MOVL C00935 V=800.0 PL=0
MOVL C00936 V=800.0 PL=0
MOVL C00937 V=800.0 PL=0
MOVL C00938 V=800.0 PL=0
MOVL C00939 V=800.0 PL=0
MOVL C00940 V=800.0 PL=0
MOVL C00941 V=800.0 PL=0
MOVL C00942 V=800.0 PL=0
MOVL C00943 V=800.0 PL=0
MOVL C00944 V=800.0 PL=0
MOVL C00945 V=800.0 PL=0
MOVL C00946 V=800.0 PL=0
MOVL C00947 V=800.0 PL=0
MOVL C00948 V=800.0 PL=0
MOVL C00949 V=800.0 PL=0
MOVL C00950 V=800.0 PL=0
MOVL C00951 V=800.0 PL=0
MOVL C00952 V=800.0 PL=0
MOVL C00953 V=800.0 PL=0
MOVL C00954 V=800.0 PL=0
MOVL C00955 V=800.0 PL=0
MOVL C00956 V=800.0 PL=0
MOVL C00957 V=800.0 PL=0
MOVL C00958 V=800.0 PL=0
MOVL C00959 V=800.0 PL=0
MOVL C00960 V=800.0 PL=0
MOVL C00961 V=800.0 PL=0
MOVL C00962 V=800.0 PL=0
MOVL C00963 V=800.0 PL=0
MOVL C00964 V=800.0 PL=0
MOVL C00965 V=800.0 PL=0
MOVL C00966 V=800.0 PL=0
MOVL C00967 V=800.0 PL=0
MOVL C00968 V=800.0 PL=0
MOVL C00969 V=800.0 PL=0
MOVL C00970 V=800.0 PL=0
MOVL C00971 V=800.0 PL=0
MOVL C00972 V=800.0 PL=0
MOVL C00973 V=800.0 PL=0
MOVL C00974 V=800.0 PL=0
MOVL C00975 V=800.0 PL=0
MOVL C00976 V=800.0 PL=0
MOVL C00977 V=800.0 PL=0
MOVL C00978 V=800.0 PL=0
MOVL C00979 V=800.0 PL=0
MOVL C00980 V=800.0 PL=0
MOVL C00981 V=800.0 PL=0
MOVL C00982 V=800.0 PL=0
MOVL C00983 V=800.0 PL=0
MOVL C00984 V=800.0 PL=0
MOVL C00985 V=800.0 PL=0
MOVL C00986 V=800.0 PL=0
MOVL C00987 V=800.0 PL=0
MOVL C00988 V=800.0 PL=0
MOVL C00989 V=800.0 PL=0
MOVL C00990 V=800.0 PL=0
MOVL C00991 V=800.0 PL=0
MOVL C00992 V=800.0 PL=0
MOVL C00993 V=800.0 PL=0
MOVL C00994 V=800.0 PL=0
MOVL C00995 V=800.0 PL=0
MOVL C00996 V=800.0 PL=0
MOVL C00997 V=800.0 PL=0
MOVL C00998 V=800.0 PL=0
MOVL C00999 V=800.0 PL=0
MOVL C01000 V=800.0 PL=0
MOVL C01001 V=800.0 PL=0
MOVL C01002 V=800.0 PL=0
MOVL C01003 V=800.0 PL=0
MOVL C01004 V=800.0 PL=0
MOVL C01005 V=800.0 PL=0
MOVL C01006 V=800.0 PL=0
MOVL C01007 V=800.0 PL=0
MOVL C01008 V=800.0 PL=0
MOVL C01009 V=800.0 PL=0
MOVL C01010 V=800.0 PL=0
MOVL C01011 V=800.0 PL=0
MOVL C01012 V=800.0 PL=0
MOVL C01013 V=800.0 PL=0
MOVL C01014 V=800.0 PL=0
MOVL C01015 V=800.0 PL=0
MOVL C01016 V=800.0 PL=0
MOVL C01017 V=800.0 PL=0
MOVL C01018 V=800.0 PL=0
MOVL C01019 V=800.0 PL=0
MOVL C01020 V=800.0 PL=0
MOVL C01021 V=800.0 PL=0
MOVL C01022 V=800.0 PL=0
MOVL C01023 V=800.0 PL=0
MOVL C01024 V=800.0 PL=0
MOVL C01025 V=800.0 PL=0
MOVL C01026 V=800.0 PL=0
MOVL C01027 V=800.0 PL=0
MOVL C01028 V=800.0 PL=0
MOVL C01029 V=800.0 PL=0
MOVL C01030 V=800.0 PL=0
MOVL C01031 V=800.0 PL=0
MOVL C01032 V=800.0 PL=0
MOVL C01033 V=800.0 PL=0
MOVL C01034 V=800.0 PL=0
MOVL C01035 V=800.0 PL=0
MOVL C01036 V=800.0 PL=0
MOVL C01037 V=800.0 PL=0
MOVL C01038 V=800.0 PL=0
MOVL C01039 V=800.0 PL=0
MOVL C01040 V=800.0 PL=0
MOVL C01041 V=800.0 PL=0
MOVL C01042 V=800.0 PL=0
MOVL C01043 V=800.0 PL=0
MOVL C01044 V=800.0 PL=0
MOVL C01045 V=800.0 PL=0
MOVL C01046 V=800.0 PL=0
MOVL C01047 V=800.0 PL=0
MOVL C01048 V=800.0 PL=0
MOVL C01049 V=800.0 PL=0
MOVL C01050 V=800.0 PL=0
MOVL C01051 V=800.0 PL=0
MOVL C01052 V=800.0 PL=0
MOVL C01053 V=800.0 PL=0
MOVL C01054 V=800.0 PL=0
MOVL C01055 V=800.0 PL=0
MOVL C01056 V=800.0 PL=0
MOVL C01057 V=800.0 PL=0
MOVL C01058 V=800.0 PL=0
MOVL C01059 V=800.0 PL=0
MOVL C01060 V=800.0 PL=0
MOVL C01061 V=800.0 PL=0
MOVL C01062 V=800.0 PL=0
MOVL C01063 V=800.0 PL=0
MOVL C01064 V=800.0 PL=0
MOVL C01065 V=800.0 PL=0
MOVL C01066 V=800.0 PL=0
MOVL C01067 V=800.0 PL=0
MOVL C01068 V=800.0 PL=0
MOVL C01069 V=800.0 PL=0
MOVL C01070 V=800.0 PL=0
MOVL C01071 V=800.0 PL=0
MOVL C01072 V=800.0 PL=0
MOVL C01073 V=800.0 PL=0
MOVL C01074 V=800.0 PL=0
MOVL C01075 V=800.0 PL=0
MOVL C01076 V=800.0 PL=0
MOVL C01077 V=800.0 PL=0
MOVL C01078 V=800.0 PL=0
MOVL C01079 V=800.0 PL=0
MOVL C01080 V=800.0 PL=0
MOVL C01081 V=800.0 PL=0
MOVL C01082 V=800.0 PL=0
MOVL C01083 V=800.0 PL=0
MOVL C01084 V=800.0 PL=0
MOVL C01085 V=800.0 PL=0
MOVL C01086 V=800.0 PL=0
MOVL C01087 V=800.0 PL=0
MOVL C01088 V=800.0 PL=0
MOVL C01089 V=800.0 PL=0
MOVL C01090 V=800.0 PL=0
MOVL C01091 V=800.0 PL=0
MOVL C01092 V=800.0 PL=0
MOVL C01093 V=800.0 PL=0
MOVL C01094 V=800.0 PL=0
MOVL C01095 V=800.0 PL=0
MOVL C01096 V=800.0 PL=0
MOVL C01097 V=800.0 PL=0
MOVL C01098 V=800.0 PL=0
MOVL C01099 V=800.0 PL=0
MOVL C01100 V=800.0 PL=0
MOVL C01101 V=800.0 PL=0
MOVL C01102 V=800.0 PL=0
MOVL C01103 V=800.0 PL=0
MOVL C01104 V=800.0 PL=0
MOVL C01105 V=800.0 PL=0
MOVL C01106 V=800.0 PL=0
MOVL C01107 V=800.0 PL=0
MOVL C01108 V=800.0 PL=0
MOVL C01109 V=800.0 PL=0
MOVL C01110 V=800.0 PL=0
MOVL C01111 V=800.0 PL=0
MOVL C01112 V=800.0 PL=0
MOVL C01113 V=800.0 PL=0
MOVL C01114 V=800.0 PL=0
MOVL C01115 V=800.0 PL=0
MOVL C01116 V=800.0 PL=0
MOVL C01117 V=800.0 PL=0
MOVL C01118 V=800.0 PL=0
MOVL C01119 V=800.0 PL=0
MOVL C01120 V=800.0 PL=0
MOVL C01121 V=800.0 PL=0
MOVL C01122 V=800.0 PL=0
MOVL C01123 V=800.0 PL=0
MOVL C01124 V=800.0 PL=0
MOVL C01125 V=800.0 PL=0
MOVL C01126 V=800.0 PL=0
MOVL C01127 V=800.0 PL=0
MOVL C01128 V=800.0 PL=0
MOVL C01129 V=800.0 PL=0
MOVL C01130 V=800.0 PL=0
MOVL C01131 V=800.0 PL=0
MOVL C01132 V=800.0 PL=0
MOVL C01133 V=800.0 PL=0
MOVL C01134 V=800.0 PL=0
MOVL C01135 V=800.0 PL=0
MOVL C01136 V=800.0 PL=0
MOVL C01137 V=800.0 PL=0
MOVL C01138 V=800.0 PL=0
MOVL C01139 V=800.0 PL=0
MOVL C01140 V=800.0 PL=0
MOVL C01141 V=800.0 PL=0
MOVL C01142 V=800.0 PL=0
MOVL C01143 V=800.0 PL=0
MOVL C01144 V=800.0 PL=0
MOVL C01145 V=800.0 PL=0
MOVL C01146 V=800.0 PL=0
MOVL C01147 V=800.0 PL=0
MOVL C01148 V=800.0 PL=0
MOVL C01149 V=800.0 PL=0
MOVL C01150 V=800.0 PL=0
MOVL C01151 V=800.0 PL=0
MOVL C01152 V=800.0 PL=0
MOVL C01153 V=800.0 PL=0
MOVL C01154 V=800.0 PL=0
MOVL C01155 V=800.0 PL=0
MOVL C01156 V=800.0 PL=0
MOVL C01157 V=800.0 PL=0
MOVL C01158 V=800.0 PL=0
MOVL C01159 V=800.0 PL=0
MOVL C01160 V=800.0 PL=0
MOVL C01161 V=800.0 PL=0
MOVL C01162 V=800.0 PL=0
MOVL C01163 V=800.0 PL=0
MOVL C01164 V=800.0 PL=0
MOVL C01165 V=800.0 PL=0
MOVL C01166 V=800.0 PL=0
MOVL C01167 V=800.0 PL=0
MOVL C01168 V=800.0 PL=0
MOVL C01169 V=800.0 PL=0
MOVL C01170 V=800.0 PL=0
MOVL C01171 V=800.0 PL=0
MOVL C01172 V=800.0 PL=0
MOVL C01173 V=800.0 PL=0
MOVL C01174 V=800.0 PL=0
MOVL C01175 V=800.0 PL=0
MOVL C01176 V=800.0 PL=0
MOVL C01177 V=800.0 PL=0
MOVL C01178 V=800.0 PL=0
MOVL C01179 V=800.0 PL=0
MOVL C01180 V=800.0 PL=0
MOVL C01181 V=800.0 PL=0
MOVL C01182 V=800.0 PL=0
MOVL C01183 V=800.0 PL=0
MOVL C01184 V=800.0 PL=0
MOVL C01185 V=800.0 PL=0
MOVL C01186 V=800.0 PL=0
MOVL C01187 V=800.0 PL=0
MOVL C01188 V=800.0 PL=0
MOVL C01189 V=800.0 PL=0
MOVL C01190 V=800.0 PL=0
MOVL C01191 V=800.0 PL=0
MOVL C01192 V=800.0 PL=0
MOVL C01193 V=800.0 PL=0
MOVL C01194 V=800.0 PL=0
MOVL C01195 V=800.0 PL=0
MOVL C01196 V=800.0 PL=0
MOVL C01197 V=800.0 PL=0
MOVL C01198 V=800.0 PL=0
MOVL C01199 V=800.0 PL=0
MOVL C01200 V=800.0 PL=0
MOVL C01201 V=800.0 PL=0
MOVL C01202 V=800.0 PL=0
MOVL C01203 V=800.0 PL=0
MOVL C01204 V=800.0 PL=0
MOVL C01205 V=800.0 PL=0
MOVL C01206 V=800.0 PL=0
MOVL C01207 V=800.0 PL=0
MOVL C01208 V=800.0 PL=0
MOVL C01209 V=800.0 PL=0
MOVL C01210 V=800.0 PL=0
MOVL C01211 V=800.0 PL=0
MOVL C01212 V=800.0 PL=0
MOVL C01213 V=800.0 PL=0
MOVL C01214 V=800.0 PL=0
MOVL C01215 V=800.0 PL=0
MOVL C01216 V=800.0 PL=0
MOVL C01217 V=800.0 PL=0
MOVL C01218 V=800.0 PL=0
MOVL C01219 V=800.0 PL=0
MOVL C01220 V=800.0 PL=0
MOVL C01221 V=800.0 PL=0
MOVL C01222 V=800.0 PL=0
MOVL C01223 V=800.0 PL=0
MOVL C01224 V=800.0 PL=0
MOVL C01225 V=800.0 PL=0
MOVL C01226 V=800.0 PL=0
MOVL C01227 V=800.0 PL=0
MOVL C01228 V=800.0 PL=0
MOVL C01229 V=800.0 PL=0
MOVL C01230 V=800.0 PL=0
MOVL C01231 V=800.0 PL=0
MOVL C01232 V=800.0 PL=0
MOVL C01233 V=800.0 PL=0
MOVL C01234 V=800.0 PL=0
MOVL C01235 V=800.0 PL=0
MOVL C01236 V=800.0 PL=0
MOVL C01237 V=800.0 PL=0
MOVL C01238 V=800.0 PL=0
MOVL C01239 V=800.0 PL=0
MOVL C01240 V=800.0 PL=0
MOVL C01241 V=800.0 PL=0
MOVL C01242 V=800.0 PL=0
MOVL C01243 V=800.0 PL=0
MOVL C01244 V=800.0 PL=0
MOVL C01245 V=800.0 PL=0
MOVL C01246 V=800.0 PL=0
MOVL C01247 V=800.0 PL=0
MOVL C01248 V=800.0 PL=0
MOVL C01249 V=800.0 PL=0
MOVL C01250 V=800.0 PL=0
MOVL C01251 V=800.0 PL=0
MOVL C01252 V=800.0 PL=0
MOVL C01253 V=800.0 PL=0
MOVL C01254 V=800.0 PL=0
MOVL C01255 V=800.0 PL=0
MOVL C01256 V=800.0 PL=0
MOVL C01257 V=800.0 PL=0
MOVL C01258 V=800.0 PL=0
MOVL C01259 V=800.0 PL=0
MOVL C01260 V=800.0 PL=0
MOVL C01261 V=800.0 PL=0
MOVL C01262 V=800.0 PL=0
MOVL C01263 V=800.0 PL=0
MOVL C01264 V=800.0 PL=0
MOVL C01265 V=800.0 PL=0
MOVL C01266 V=800.0 PL=0
MOVL C01267 V=800.0 PL=0
MOVL C01268 V=800.0 PL=0
MOVL C01269 V=800.0 PL=0
MOVL C01270 V=800.0 PL=0
MOVL C01271 V=800.0 PL=0
MOVL C01272 V=800.0 PL=0
MOVL C01273 V=800.0 PL=0
MOVL C01274 V=800.0 PL=0
MOVL C01275 V=800.0 PL=0
MOVL C01276 V=800.0 PL=0
MOVL C01277 V=800.0 PL=0
MOVL C01278 V=800.0 PL=0
MOVL C01279 V=800.0 PL=0
MOVL C01280 V=800.0 PL=0
MOVL C01281 V=800.0 PL=0
MOVL C01282 V=800.0 PL=0
MOVL C01283 V=800.0 PL=0
MOVL C01284 V=800.0 PL=0
MOVL C01285 V=800.0 PL=0
MOVL C01286 V=800.0 PL=0
MOVL C01287 V=800.0 PL=0
MOVL C01288 V=800.0 PL=0
MOVL C01289 V=800.0 PL=0
MOVL C01290 V=800.0 PL=0
MOVL C01291 V=800.0 PL=0
MOVL C01292 V=800.0 PL=0
MOVL C01293 V=800.0 PL=0
MOVL C01294 V=800.0 PL=0
MOVL C01295 V=800.0 PL=0
MOVL C01296 V=800.0 PL=0
MOVL C01297 V=800.0 PL=0
MOVL C01298 V=800.0 PL=0
MOVL C01299 V=800.0 PL=0
MOVL C01300 V=800.0 PL=0
MOVL C01301 V=800.0 PL=0
MOVL C01302 V=800.0 PL=0
MOVL C01303 V=800.0 PL=0
MOVL C01304 V=800.0 PL=0
MOVL C01305 V=800.0 PL=0
MOVL C01306 V=800.0 PL=0
MOVL C01307 V=800.0 PL=0
MOVL C01308 V=800.0 PL=0
MOVL C01309 V=800.0 PL=0
MOVL C01310 V=800.0 PL=0
MOVL C01311 V=800.0 PL=0
MOVL C01312 V=800.0 PL=0
MOVL C01313 V=800.0 PL=0
MOVL C01314 V=800.0 PL=0
MOVL C01315 V=800.0 PL=0
MOVL C01316 V=800.0 PL=0
MOVL C01317 V=800.0 PL=0
MOVL C01318 V=800.0 PL=0
MOVL C01319 V=800.0 PL=0
MOVL C01320 V=800.0 PL=0
MOVL C01321 V=800.0 PL=0
MOVL C01322 V=800.0 PL=0
MOVL C01323 V=800.0 PL=0
MOVL C01324 V=800.0 PL=0
MOVL C01325 V=800.0 PL=0
MOVL C01326 V=800.0 PL=0
MOVL C01327 V=800.0 PL=0
MOVL C01328 V=800.0 PL=0
MOVL C01329 V=800.0 PL=0
MOVL C01330 V=800.0 PL=0
MOVL C01331 V=800.0 PL=0
MOVL C01332 V=800.0 PL=0
MOVL C01333 V=800.0 PL=0
MOVL C01334 V=800.0 PL=0
MOVL C01335 V=800.0 PL=0
MOVL C01336 V=800.0 PL=0
MOVL C01337 V=800.0 PL=0
MOVL C01338 V=800.0 PL=0
MOVL C01339 V=800.0 PL=0
MOVL C01340 V=800.0 PL=0
MOVL C01341 V=800.0 PL=0
MOVL C01342 V=800.0 PL=0
MOVL C01343 V=800.0 PL=0
MOVL C01344 V=800.0 PL=0
MOVL C01345 V=800.0 PL=0
MOVL C01346 V=800.0 PL=0
MOVL C01347 V=800.0 PL=0
MOVL C01348 V=800.0 PL=0
MOVL C01349 V=800.0 PL=0
MOVL C01350 V=800.0 PL=0
MOVL C01351 V=800.0 PL=0
MOVL C01352 V=800.0 PL=0
MOVL C01353 V=800.0 PL=0
MOVL C01354 V=800.0 PL=0
MOVL C01355 V=800.0 PL=0
MOVL C01356 V=800.0 PL=0
MOVL C01357 V=800.0 PL=0
MOVL C01358 V=800.0 PL=0
MOVL C01359 V=800.0 PL=0
MOVL C01360 V=800.0 PL=0
MOVL C01361 V=800.0 PL=0
MOVL C01362 V=800.0 PL=0
MOVL C01363 V=800.0 PL=0
MOVL C01364 V=800.0 PL=0
MOVL C01365 V=800.0 PL=0
MOVL C01366 V=800.0 PL=0
MOVL C01367 V=800.0 PL=0
MOVL C01368 V=800.0 PL=0
MOVL C01369 V=800.0 PL=0
MOVL C01370 V=800.0 PL=0
MOVL C01371 V=800.0 PL=0
MOVL C01372 V=800.0 PL=0
MOVL C01373 V=800.0 PL=0
MOVL C01374 V=800.0 PL=0
MOVL C01375 V=800.0 PL=0
MOVL C01376 V=800.0 PL=0
MOVL C01377 V=800.0 PL=0
MOVL C01378 V=800.0 PL=0
MOVL C01379 V=800.0 PL=0
MOVL C01380 V=800.0 PL=0
MOVL C01381 V=800.0 PL=0
MOVL C01382 V=800.0 PL=0
MOVL C01383 V=800.0 PL=0
MOVL C01384 V=800.0 PL=0
MOVL C01385 V=800.0 PL=0
MOVL C01386 V=800.0 PL=0
MOVL C01387 V=800.0 PL=0
MOVL C01388 V=800.0 PL=0
MOVL C01389 V=800.0 PL=0
MOVL C01390 V=800.0 PL=0
MOVL C01391 V=800.0 PL=0
MOVL C01392 V=800.0 PL=0
MOVL C01393 V=800.0 PL=0
MOVL C01394 V=800.0 PL=0
MOVL C01395 V=800.0 PL=0
MOVL C01396 V=800.0 PL=0
MOVL C01397 V=800.0 PL=0
MOVL C01398 V=800.0 PL=0
MOVL C01399 V=800.0 PL=0
MOVL C01400 V=800.0 PL=0
MOVL C01401 V=800.0 PL=0
MOVL C01402 V=800.0 PL=0
MOVL C01403 V=800.0 PL=0
MOVL C01404 V=800.0 PL=0
MOVL C01405 V=800.0 PL=0
MOVL C01406 V=800.0 PL=0
MOVL C01407 V=800.0 PL=0
MOVL C01408 V=800.0 PL=0
MOVL C01409 V=800.0 PL=0
MOVL C01410 V=800.0 PL=0
MOVL C01411 V=800.0 PL=0
MOVL C01412 V=800.0 PL=0
MOVL C01413 V=800.0 PL=0
MOVL C01414 V=800.0 PL=0
MOVL C01415 V=800.0 PL=0
MOVL C01416 V=800.0 PL=0
MOVL C01417 V=800.0 PL=0
MOVL C01418 V=800.0 PL=0
MOVL C01419 V=800.0 PL=0
MOVL C01420 V=800.0 PL=0
MOVL C01421 V=800.0 PL=0
MOVL C01422 V=800.0 PL=0
MOVL C01423 V=800.0 PL=0
MOVL C01424 V=800.0 PL=0
MOVL C01425 V=800.0 PL=0
MOVL C01426 V=800.0 PL=0
MOVL C01427 V=800.0 PL=0
MOVL C01428 V=800.0 PL=0
MOVL C01429 V=800.0 PL=0
MOVL C01430 V=800.0 PL=0
MOVL C01431 V=800.0 PL=0
MOVL C01432 V=800.0 PL=0
MOVL C01433 V=800.0 PL=0
MOVL C01434 V=800.0 PL=0
MOVL C01435 V=800.0 PL=0
MOVL C01436 V=800.0 PL=0
MOVL C01437 V=800.0 PL=0
MOVL C01438 V=800.0 PL=0
MOVL C01439 V=800.0 PL=0
MOVL C01440 V=800.0 PL=0
MOVL C01441 V=800.0 PL=0
MOVL C01442 V=800.0 PL=0
MOVL C01443 V=800.0 PL=0
MOVL C01444 V=800.0 PL=0
MOVL C01445 V=800.0 PL=0
MOVL C01446 V=800.0 PL=0
MOVL C01447 V=800.0 PL=0
MOVL C01448 V=800.0 PL=0
MOVL C01449 V=800.0 PL=0
MOVL C01450 V=800.0 PL=0
MOVL C01451 V=800.0 PL=0
MOVL C01452 V=800.0 PL=0
MOVL C01453 V=800.0 PL=0
MOVL C01454 V=800.0 PL=0
MOVL C01455 V=800.0 PL=0
MOVL C01456 V=800.0 PL=0
MOVL C01457 V=800.0 PL=0
MOVL C01458 V=800.0 PL=0
MOVL C01459 V=800.0 PL=0
MOVL C01460 V=800.0 PL=0
MOVL C01461 V=800.0 PL=0
MOVL C01462 V=800.0 PL=0
MOVL C01463 V=800.0 PL=0
MOVL C01464 V=800.0 PL=0
MOVL C01465 V=800.0 PL=0
MOVL C01466 V=800.0 PL=0
MOVL C01467 V=800.0 PL=0
MOVL C01468 V=800.0 PL=0
MOVL C01469 V=800.0 PL=0
MOVL C01470 V=800.0 PL=0
MOVL C01471 V=800.0 PL=0
MOVL C01472 V=800.0 PL=0
MOVL C01473 V=800.0 PL=0
MOVL C01474 V=800.0 PL=0
MOVL C01475 V=800.0 PL=0
MOVL C01476 V=800.0 PL=0
MOVL C01477 V=800.0 PL=0
MOVL C01478 V=800.0 PL=0
MOVL C01479 V=800.0 PL=0
MOVL C01480 V=800.0 PL=0
MOVL C01481 V=800.0 PL=0
MOVL C01482 V=800.0 PL=0
MOVL C01483 V=800.0 PL=0
MOVL C01484 V=800.0 PL=0
MOVL C01485 V=800.0 PL=0
MOVL C01486 V=800.0 PL=0
MOVL C01487 V=800.0 PL=0
MOVL C01488 V=800.0 PL=0
MOVL C01489 V=800.0 PL=0
MOVL C01490 V=800.0 PL=0
MOVL C01491 V=800.0 PL=0
MOVL C01492 V=800.0 PL=0
MOVL C01493 V=800.0 PL=0
MOVL C01494 V=800.0 PL=0
MOVL C01495 V=800.0 PL=0
MOVL C01496 V=800.0 PL=0
MOVL C01497 V=800.0 PL=0
MOVL C01498 V=800.0 PL=0
MOVL C01499 V=800.0 PL=0
MOVL C01500 V=800.0 PL=0
MOVL C01501 V=800.0 PL=0
MOVL C01502 V=800.0 PL=0
MOVL C01503 V=800.0 PL=0
MOVL C01504 V=800.0 PL=0
MOVL C01505 V=800.0 PL=0
MOVL C01506 V=800.0 PL=0
MOVL C01507 V=800.0 PL=0
MOVL C01508 V=800.0 PL=0
MOVL C01509 V=800.0 PL=0
MOVL C01510 V=800.0 PL=0
MOVL C01511 V=800.0 PL=0
MOVL C01512 V=800.0 PL=0
MOVL C01513 V=800.0 PL=0
MOVL C01514 V=800.0 PL=0
MOVL C01515 V=800.0 PL=0
MOVL C01516 V=800.0 PL=0
MOVL C01517 V=800.0 PL=0
MOVL C01518 V=800.0 PL=0
MOVL C01519 V=800.0 PL=0
MOVL C01520 V=800.0 PL=0
MOVL C01521 V=800.0 PL=0
MOVL C01522 V=800.0 PL=0
MOVL C01523 V=800.0 PL=0
MOVL C01524 V=800.0 PL=0
MOVL C01525 V=800.0 PL=0
MOVL C01526 V=800.0 PL=0
MOVL C01527 V=800.0 PL=0
MOVL C01528 V=800.0 PL=0
MOVL C01529 V=800.0 PL=0
MOVL C01530 V=800.0 PL=0
MOVL C01531 V=800.0 PL=0
MOVL C01532 V=800.0 PL=0
MOVL C01533 V=800.0 PL=0
MOVL C01534 V=800.0 PL=0
MOVL C01535 V=800.0 PL=0
MOVL C01536 V=800.0 PL=0
MOVL C01537 V=800.0 PL=0
MOVL C01538 V=800.0 PL=0
MOVL C01539 V=800.0 PL=0
MOVL C01540 V=800.0 PL=0
MOVL C01541 V=800.0 PL=0
MOVL C01542 V=800.0 PL=0
MOVL C01543 V=800.0 PL=0
MOVL C01544 V=800.0 PL=0
MOVL C01545 V=800.0 PL=0
MOVL C01546 V=800.0 PL=0
MOVL C01547 V=800.0 PL=0
MOVL C01548 V=800.0 PL=0
MOVL C01549 V=800.0 PL=0
MOVL C01550 V=800.0 PL=0
MOVL C01551 V=800.0 PL=0
MOVL C01552 V=800.0 PL=0
MOVL C01553 V=800.0 PL=0
MOVL C01554 V=800.0 PL=0
MOVL C01555 V=800.0 PL=0
MOVL C01556 V=800.0 PL=0
MOVL C01557 V=800.0 PL=0
MOVL C01558 V=800.0 PL=0
MOVL C01559 V=800.0 PL=0
MOVL C01560 V=800.0 PL=0
MOVL C01561 V=800.0 PL=0
MOVL C01562 V=800.0 PL=0
MOVL C01563 V=800.0 PL=0
MOVL C01564 V=800.0 PL=0
MOVL C01565 V=800.0 PL=0
MOVL C01566 V=800.0 PL=0
MOVL C01567 V=800.0 PL=0
MOVL C01568 V=800.0 PL=0
MOVL C01569 V=800.0 PL=0
MOVL C01570 V=800.0 PL=0
MOVL C01571 V=800.0 PL=0
MOVL C01572 V=800.0 PL=0
MOVL C01573 V=800.0 PL=0
MOVL C01574 V=800.0 PL=0
MOVL C01575 V=800.0 PL=0
MOVL C01576 V=800.0 PL=0
MOVL C01577 V=800.0 PL=0
MOVL C01578 V=800.0 PL=0
MOVL C01579 V=800.0 PL=0
MOVL C01580 V=800.0 PL=0
MOVL C01581 V=800.0 PL=0
MOVL C01582 V=800.0 PL=0
MOVL C01583 V=800.0 PL=0
MOVL C01584 V=800.0 PL=0
MOVL C01585 V=800.0 PL=0
MOVL C01586 V=800.0 PL=0
MOVL C01587 V=800.0 PL=0
MOVL C01588 V=800.0 PL=0
MOVL C01589 V=800.0 PL=0
MOVL C01590 V=800.0 PL=0
MOVL C01591 V=800.0 PL=0
MOVL C01592 V=800.0 PL=0
MOVL C01593 V=800.0 PL=0
MOVL C01594 V=800.0 PL=0
MOVL C01595 V=800.0 PL=0
MOVL C01596 V=800.0 PL=0
MOVL C01597 V=800.0 PL=0
MOVL C01598 V=800.0 PL=0
MOVL C01599 V=800.0 PL=0
MOVL C01600 V=800.0 PL=0
MOVL C01601 V=800.0 PL=0
MOVL C01602 V=800.0 PL=0
MOVL C01603 V=800.0 PL=0
MOVL C01604 V=800.0 PL=0
MOVL C01605 V=800.0 PL=0
MOVL C01606 V=800.0 PL=0
MOVL C01607 V=800.0 PL=0
MOVL C01608 V=800.0 PL=0
MOVL C01609 V=800.0 PL=0
MOVL C01610 V=800.0 PL=0
MOVL C01611 V=800.0 PL=0
MOVL C01612 V=800.0 PL=0
MOVL C01613 V=800.0 PL=0
MOVL C01614 V=800.0 PL=0
MOVL C01615 V=800.0 PL=0
MOVL C01616 V=800.0 PL=0
MOVL C01617 V=800.0 PL=0
MOVL C01618 V=800.0 PL=0
MOVL C01619 V=800.0 PL=0
MOVL C01620 V=800.0 PL=0
MOVL C01621 V=800.0 PL=0
MOVL C01622 V=800.0 PL=0
MOVL C01623 V=800.0 PL=0
MOVL C01624 V=800.0 PL=0
MOVL C01625 V=800.0 PL=0
MOVL C01626 V=800.0 PL=0
MOVL C01627 V=800.0 PL=0
MOVL C01628 V=800.0 PL=0
MOVL C01629 V=800.0 PL=0
MOVL C01630 V=800.0 PL=0
MOVL C01631 V=800.0 PL=0
MOVL C01632 V=800.0 PL=0
MOVL C01633 V=800.0 PL=0
MOVL C01634 V=800.0 PL=0
MOVL C01635 V=800.0 PL=0
MOVL C01636 V=800.0 PL=0
MOVL C01637 V=800.0 PL=0
MOVL C01638 V=800.0 PL=0
MOVL C01639 V=800.0 PL=0
MOVL C01640 V=800.0 PL=0
MOVL C01641 V=800.0 PL=0
MOVL C01642 V=800.0 PL=0
MOVL C01643 V=800.0 PL=0
MOVL C01644 V=800.0 PL=0
MOVL C01645 V=800.0 PL=0
MOVL C01646 V=800.0 PL=0
MOVL C01647 V=800.0 PL=0
MOVL C01648 V=800.0 PL=0
MOVL C01649 V=800.0 PL=0
MOVL C01650 V=800.0 PL=0
MOVL C01651 V=800.0 PL=0
MOVL C01652 V=800.0 PL=0
MOVL C01653 V=800.0 PL=0
MOVL C01654 V=800.0 PL=0
MOVL C01655 V=800.0 PL=0
MOVL C01656 V=800.0 PL=0
MOVL C01657 V=800.0 PL=0
MOVL C01658 V=800.0 PL=0
MOVL C01659 V=800.0 PL=0
MOVL C01660 V=800.0 PL=0
MOVL C01661 V=800.0 PL=0
MOVL C01662 V=800.0 PL=0
MOVL C01663 V=800.0 PL=0
MOVL C01664 V=800.0 PL=0
MOVL C01665 V=800.0 PL=0
MOVL C01666 V=800.0 PL=0
MOVL C01667 V=800.0 PL=0
MOVL C01668 V=800.0 PL=0
MOVL C01669 V=800.0 PL=0
MOVL C01670 V=800.0 PL=0
MOVL C01671 V=800.0 PL=0
MOVL C01672 V=800.0 PL=0
MOVL C01673 V=800.0 PL=0
MOVL C01674 V=800.0 PL=0
MOVL C01675 V=800.0 PL=0
MOVL C01676 V=800.0 PL=0
MOVL C01677 V=800.0 PL=0
MOVL C01678 V=800.0 PL=0
MOVL C01679 V=800.0 PL=0
MOVL C01680 V=800.0 PL=0
MOVL C01681 V=800.0 PL=0
MOVL C01682 V=800.0 PL=0
MOVL C01683 V=800.0 PL=0
MOVL C01684 V=800.0 PL=0
MOVL C01685 V=800.0 PL=0
MOVL C01686 V=800.0 PL=0
MOVL C01687 V=800.0 PL=0
MOVL C01688 V=800.0 PL=0
MOVL C01689 V=800.0 PL=0
MOVL C01690 V=800.0 PL=0
MOVL C01691 V=800.0 PL=0
MOVL C01692 V=800.0 PL=0
MOVL C01693 V=800.0 PL=0
MOVL C01694 V=800.0 PL=0
MOVL C01695 V=800.0 PL=0
MOVL C01696 V=800.0 PL=0
MOVL C01697 V=800.0 PL=0
MOVL C01698 V=800.0 PL=0
MOVL C01699 V=800.0 PL=0
MOVL C01700 V=800.0 PL=0
MOVL C01701 V=800.0 PL=0
MOVL C01702 V=800.0 PL=0
MOVL C01703 V=800.0 PL=0
MOVL C01704 V=800.0 PL=0
MOVL C01705 V=800.0 PL=0
MOVL C01706 V=800.0 PL=0
MOVL C01707 V=800.0 PL=0
MOVL C01708 V=800.0 PL=0
MOVL C01709 V=800.0 PL=0
MOVL C01710 V=800.0 PL=0
MOVL C01711 V=800.0 PL=0
MOVL C01712 V=800.0 PL=0
MOVL C01713 V=800.0 PL=0
MOVL C01714 V=800.0 PL=0
MOVL C01715 V=800.0 PL=0
MOVL C01716 V=800.0 PL=0
MOVL C01717 V=800.0 PL=0
MOVL C01718 V=800.0 PL=0
MOVL C01719 V=800.0 PL=0
MOVL C01720 V=800.0 PL=0
MOVL C01721 V=800.0 PL=0
MOVL C01722 V=800.0 PL=0
MOVL C01723 V=800.0 PL=0
MOVL C01724 V=800.0 PL=0
MOVL C01725 V=800.0 PL=0
MOVL C01726 V=800.0 PL=0
MOVL C01727 V=800.0 PL=0
MOVL C01728 V=800.0 PL=0
MOVL C01729 V=800.0 PL=0
MOVL C01730 V=800.0 PL=0
MOVL C01731 V=800.0 PL=0
MOVL C01732 V=800.0 PL=0
MOVL C01733 V=800.0 PL=0
MOVL C01734 V=800.0 PL=0
MOVL C01735 V=800.0 PL=0
MOVL C01736 V=800.0 PL=0
MOVL C01737 V=800.0 PL=0
MOVL C01738 V=800.0 PL=0
MOVL C01739 V=800.0 PL=0
MOVL C01740 V=800.0 PL=0
MOVL C01741 V=800.0 PL=0
MOVL C01742 V=800.0 PL=0
MOVL C01743 V=800.0 PL=0
MOVL C01744 V=800.0 PL=0
MOVL C01745 V=800.0 PL=0
MOVL C01746 V=800.0 PL=0
MOVL C01747 V=800.0 PL=0
MOVL C01748 V=800.0 PL=0
MOVL C01749 V=800.0 PL=0
MOVL C01750 V=800.0 PL=0
MOVL C01751 V=800.0 PL=0
MOVL C01752 V=800.0 PL=0
MOVL C01753 V=800.0 PL=0
MOVL C01754 V=800.0 PL=0
MOVL C01755 V=800.0 PL=0
MOVL C01756 V=800.0 PL=0
MOVL C01757 V=800.0 PL=0
MOVL C01758 V=800.0 PL=0
MOVL C01759 V=800.0 PL=0
MOVL C01760 V=800.0 PL=0
MOVL C01761 V=800.0 PL=0
MOVL C01762 V=800.0 PL=0
MOVL C01763 V=800.0 PL=0
MOVL C01764 V=800.0 PL=0
MOVL C01765 V=800.0 PL=0
MOVL C01766 V=800.0 PL=0
MOVL C01767 V=800.0 PL=0
MOVL C01768 V=800.0 PL=0
MOVL C01769 V=800.0 PL=0
MOVL C01770 V=800.0 PL=0
MOVL C01771 V=800.0 PL=0
MOVL C01772 V=800.0 PL=0
MOVL C01773 V=800.0 PL=0
MOVL C01774 V=800.0 PL=0
MOVL C01775 V=800.0 PL=0
MOVL C01776 V=800.0 PL=0
MOVL C01777 V=800.0 PL=0
MOVL C01778 V=800.0 PL=0
MOVL C01779 V=800.0 PL=0
MOVL C01780 V=800.0 PL=0
MOVL C01781 V=800.0 PL=0
MOVL C01782 V=800.0 PL=0
MOVL C01783 V=800.0 PL=0
MOVL C01784 V=800.0 PL=0
MOVL C01785 V=800.0 PL=0
MOVL C01786 V=800.0 PL=0
MOVL C01787 V=800.0 PL=0
MOVL C01788 V=800.0 PL=0
MOVL C01789 V=800.0 PL=0
MOVL C01790 V=800.0 PL=0
MOVL C01791 V=800.0 PL=0
MOVL C01792 V=800.0 PL=0
MOVL C01793 V=800.0 PL=0
MOVL C01794 V=800.0 PL=0
MOVL C01795 V=800.0 PL=0
MOVL C01796 V=800.0 PL=0
MOVL C01797 V=800.0 PL=0
MOVL C01798 V=800.0 PL=0
MOVL C01799 V=800.0 PL=0
MOVL C01800 V=800.0 PL=0
MOVL C01801 V=800.0 PL=0
MOVL C01802 V=800.0 PL=0
MOVL C01803 V=800.0 PL=0
MOVL C01804 V=800.0 PL=0
MOVL C01805 V=800.0 PL=0
MOVL C01806 V=800.0 PL=0
MOVL C01807 V=800.0 PL=0
MOVL C01808 V=800.0 PL=0
MOVL C01809 V=800.0 PL=0
MOVL C01810 V=800.0 PL=0
MOVL C01811 V=800.0 PL=0
MOVL C01812 V=800.0 PL=0
MOVL C01813 V=800.0 PL=0
MOVL C01814 V=800.0 PL=0
MOVL C01815 V=800.0 PL=0
MOVL C01816 V=800.0 PL=0
MOVL C01817 V=800.0 PL=0
MOVL C01818 V=800.0 PL=0
MOVL C01819 V=800.0 PL=0
MOVL C01820 V=800.0 PL=0
MOVL C01821 V=800.0 PL=0
MOVL C01822 V=800.0 PL=0
MOVL C01823 V=800.0 PL=0
MOVL C01824 V=800.0 PL=0
MOVL C01825 V=800.0 PL=0
MOVL C01826 V=800.0 PL=0
MOVL C01827 V=800.0 PL=0
MOVL C01828 V=800.0 PL=0
MOVL C01829 V=800.0 PL=0
MOVL C01830 V=800.0 PL=0
MOVL C01831 V=800.0 PL=0
MOVL C01832 V=800.0 PL=0
MOVL C01833 V=800.0 PL=0
MOVL C01834 V=800.0 PL=0
MOVL C01835 V=800.0 PL=0
MOVL C01836 V=800.0 PL=0
MOVL C01837 V=800.0 PL=0
MOVL C01838 V=800.0 PL=0
MOVL C01839 V=800.0 PL=0
MOVL C01840 V=800.0 PL=0
MOVL C01841 V=800.0 PL=0
MOVL C01842 V=800.0 PL=0
MOVL C01843 V=800.0 PL=0
MOVL C01844 V=800.0 PL=0
MOVL C01845 V=800.0 PL=0
MOVL C01846 V=800.0 PL=0
MOVL C01847 V=800.0 PL=0
MOVL C01848 V=800.0 PL=0
MOVL C01849 V=800.0 PL=0
MOVL C01850 V=800.0 PL=0
MOVL C01851 V=800.0 PL=0
MOVL C01852 V=800.0 PL=0
MOVL C01853 V=800.0 PL=0
MOVL C01854 V=800.0 PL=0
MOVL C01855 V=800.0 PL=0
MOVL C01856 V=800.0 PL=0
MOVL C01857 V=800.0 PL=0
MOVL C01858 V=800.0 PL=0
MOVL C01859 V=800.0 PL=0
MOVL C01860 V=800.0 PL=0
MOVL C01861 V=800.0 PL=0
MOVL C01862 V=800.0 PL=0
MOVL C01863 V=800.0 PL=0
MOVL C01864 V=800.0 PL=0
MOVL C01865 V=800.0 PL=0
MOVL C01866 V=800.0 PL=0
MOVL C01867 V=800.0 PL=0
MOVL C01868 V=800.0 PL=0
MOVL C01869 V=800.0 PL=0
MOVL C01870 V=800.0 PL=0
MOVL C01871 V=800.0 PL=0
MOVL C01872 V=800.0 PL=0
MOVL C01873 V=800.0 PL=0
MOVL C01874 V=800.0 PL=0
MOVL C01875 V=800.0 PL=0
MOVL C01876 V=800.0 PL=0
MOVL C01877 V=800.0 PL=0
MOVL C01878 V=800.0 PL=0
MOVL C01879 V=800.0 PL=0
MOVL C01880 V=800.0 PL=0
MOVL C01881 V=800.0 PL=0
MOVL C01882 V=800.0 PL=0
MOVL C01883 V=800.0 PL=0
MOVL C01884 V=800.0 PL=0
MOVL C01885 V=800.0 PL=0
MOVL C01886 V=800.0 PL=0
MOVL C01887 V=800.0 PL=0
MOVL C01888 V=800.0 PL=0
MOVL C01889 V=800.0 PL=0
MOVL C01890 V=800.0 PL=0
MOVL C01891 V=800.0 PL=0
MOVL C01892 V=800.0 PL=0
MOVL C01893 V=800.0 PL=0
MOVL C01894 V=800.0 PL=0
MOVL C01895 V=800.0 PL=0
MOVL C01896 V=800.0 PL=0
MOVL C01897 V=800.0 PL=0
MOVL C01898 V=800.0 PL=0
MOVL C01899 V=800.0 PL=0
MOVL C01900 V=800.0 PL=0
MOVL C01901 V=800.0 PL=0
MOVL C01902 V=800.0 PL=0
MOVL C01903 V=800.0 PL=0
MOVL C01904 V=800.0 PL=0
MOVL C01905 V=800.0 PL=0
MOVL C01906 V=800.0 PL=0
MOVL C01907 V=800.0 PL=0
MOVL C01908 V=800.0 PL=0
MOVL C01909 V=800.0 PL=0
MOVL C01910 V=800.0 PL=0
MOVL C01911 V=800.0 PL=0
MOVL C01912 V=800.0 PL=0
MOVL C01913 V=800.0 PL=0
MOVL C01914 V=800.0 PL=0
MOVL C01915 V=800.0 PL=0
MOVL C01916 V=800.0 PL=0
MOVL C01917 V=800.0 PL=0
MOVL C01918 V=800.0 PL=0
MOVL C01919 V=800.0 PL=0
MOVL C01920 V=800.0 PL=0
MOVL C01921 V=800.0 PL=0
MOVL C01922 V=800.0 PL=0
MOVL C01923 V=800.0 PL=0
MOVL C01924 V=800.0 PL=0
MOVL C01925 V=800.0 PL=0
MOVL C01926 V=800.0 PL=0
MOVL C01927 V=800.0 PL=0
MOVL C01928 V=800.0 PL=0
MOVL C01929 V=800.0 PL=0
MOVL C01930 V=800.0 PL=0
MOVL C01931 V=800.0 PL=0
MOVL C01932 V=800.0 PL=0
MOVL C01933 V=800.0 PL=0
MOVL C01934 V=800.0 PL=0
MOVL C01935 V=800.0 PL=0
MOVL C01936 V=800.0 PL=0
MOVL C01937 V=800.0 PL=0
MOVL C01938 V=800.0 PL=0
MOVL C01939 V=800.0 PL=0
MOVL C01940 V=800.0 PL=0
MOVL C01941 V=800.0 PL=0
MOVL C01942 V=800.0 PL=0
MOVL C01943 V=800.0 PL=0
MOVL C01944 V=800.0 PL=0
MOVL C01945 V=800.0 PL=0
MOVL C01946 V=800.0 PL=0
MOVL C01947 V=800.0 PL=0
MOVL C01948 V=800.0 PL=0
MOVL C01949 V=800.0 PL=0
MOVL C01950 V=800.0 PL=0
MOVL C01951 V=800.0 PL=0
MOVL C01952 V=800.0 PL=0
MOVL C01953 V=800.0 PL=0
MOVL C01954 V=800.0 PL=0
MOVL C01955 V=800.0 PL=0
MOVL C01956 V=800.0 PL=0
MOVL C01957 V=800.0 PL=0
MOVL C01958 V=800.0 PL=0
MOVL C01959 V=800.0 PL=0
MOVL C01960 V=800.0 PL=0
MOVL C01961 V=800.0 PL=0
MOVL C01962 V=800.0 PL=0
MOVL C01963 V=800.0 PL=0
MOVL C01964 V=800.0 PL=0
MOVL C01965 V=800.0 PL=0
MOVL C01966 V=800.0 PL=0
MOVL C01967 V=800.0 PL=0
MOVL C01968 V=800.0 PL=0
MOVL C01969 V=800.0 PL=0
MOVL C01970 V=800.0 PL=0
MOVL C01971 V=800.0 PL=0
MOVL C01972 V=800.0 PL=0
MOVL C01973 V=800.0 PL=0
MOVL C01974 V=800.0 PL=0
MOVL C01975 V=800.0 PL=0
MOVL C01976 V=800.0 PL=0
MOVL C01977 V=800.0 PL=0
MOVL C01978 V=800.0 PL=0
MOVL C01979 V=800.0 PL=0
MOVL C01980 V=800.0 PL=0
MOVL C01981 V=800.0 PL=0
MOVL C01982 V=800.0 PL=0
MOVL C01983 V=800.0 PL=0
MOVL C01984 V=800.0 PL=0
MOVL C01985 V=800.0 PL=0
MOVL C01986 V=800.0 PL=0
MOVL C01987 V=800.0 PL=0
MOVL C01988 V=800.0 PL=0
MOVL C01989 V=800.0 PL=0
MOVL C01990 V=800.0 PL=0
MOVL C01991 V=800.0 PL=0
MOVL C01992 V=800.0 PL=0
MOVL C01993 V=800.0 PL=0
MOVL C01994 V=800.0 PL=0
MOVL C01995 V=800.0 PL=0
MOVL C01996 V=800.0 PL=0
MOVL C01997 V=800.0 PL=0
MOVL C01998 V=800.0 PL=0
MOVL C01999 V=800.0 PL=0
MOVL C02000 V=800.0 PL=0
MOVL C02001 V=800.0 PL=0
MOVL C02002 V=800.0 PL=0
MOVL C02003 V=800.0 PL=0
MOVL C02004 V=800.0 PL=0
MOVL C02005 V=800.0 PL=0
MOVL C02006 V=800.0 PL=0
MOVL C02007 V=800.0 PL=0
MOVL C02008 V=800.0 PL=0
MOVL C02009 V=800.0 PL=0
MOVL C02010 V=800.0 PL=0
MOVL C02011 V=800.0 PL=0
MOVL C02012 V=800.0 PL=0
MOVL C02013 V=800.0 PL=0
MOVL C02014 V=800.0 PL=0
MOVL C02015 V=800.0 PL=0
MOVL C02016 V=800.0 PL=0
MOVL C02017 V=800.0 PL=0
MOVL C02018 V=800.0 PL=0
MOVL C02019 V=800.0 PL=0
MOVL C02020 V=800.0 PL=0
MOVL C02021 V=800.0 PL=0
MOVL C02022 V=800.0 PL=0
MOVL C02023 V=800.0 PL=0
MOVL C02024 V=800.0 PL=0
MOVL C02025 V=800.0 PL=0
MOVL C02026 V=800.0 PL=0
MOVL C02027 V=800.0 PL=0
MOVL C02028 V=800.0 PL=0
MOVL C02029 V=800.0 PL=0
MOVL C02030 V=800.0 PL=0
MOVL C02031 V=800.0 PL=0
MOVL C02032 V=800.0 PL=0
MOVL C02033 V=800.0 PL=0
MOVL C02034 V=800.0 PL=0
MOVL C02035 V=800.0 PL=0
MOVL C02036 V=800.0 PL=0
MOVL C02037 V=800.0 PL=0
MOVL C02038 V=800.0 PL=0
MOVL C02039 V=800.0 PL=0
MOVL C02040 V=800.0 PL=0
MOVL C02041 V=800.0 PL=0
MOVL C02042 V=800.0 PL=0
MOVL C02043 V=800.0 PL=0
MOVL C02044 V=800.0 PL=0
MOVL C02045 V=800.0 PL=0
MOVL C02046 V=800.0 PL=0
MOVL C02047 V=800.0 PL=0
MOVL C02048 V=800.0 PL=0
MOVL C02049 V=800.0 PL=0
MOVL C02050 V=800.0 PL=0
MOVL C02051 V=800.0 PL=0
MOVL C02052 V=800.0 PL=0
MOVL C02053 V=800.0 PL=0
MOVL C02054 V=800.0 PL=0
MOVL C02055 V=800.0 PL=0
MOVL C02056 V=800.0 PL=0
MOVL C02057 V=800.0 PL=0
MOVL C02058 V=800.0 PL=0
MOVL C02059 V=800.0 PL=0
MOVL C02060 V=800.0 PL=0
MOVL C02061 V=800.0 PL=0
MOVL C02062 V=800.0 PL=0
MOVL C02063 V=800.0 PL=0
MOVL C02064 V=800.0 PL=0
MOVL C02065 V=800.0 PL=0
MOVL C02066 V=800.0 PL=0
MOVL C02067 V=800.0 PL=0
MOVL C02068 V=800.0 PL=0
MOVL C02069 V=800.0 PL=0
MOVL C02070 V=800.0 PL=0
MOVL C02071 V=800.0 PL=0
MOVL C02072 V=800.0 PL=0
MOVL C02073 V=800.0 PL=0
MOVL C02074 V=800.0 PL=0
MOVL C02075 V=800.0 PL=0
MOVL C02076 V=800.0 PL=0
MOVL C02077 V=800.0 PL=0
MOVL C02078 V=800.0 PL=0
MOVL C02079 V=800.0 PL=0
MOVL C02080 V=800.0 PL=0
MOVL C02081 V=800.0 PL=0
